VAR_INPUT
  VALUE : TIME_OF_DAY ;	//Zu prüfender Wert
  MIN : TIME_OF_DAY ;	//Zulässiger Minimalwert
  MAX : TIME_OF_DAY ;	//Zulässiger Maximalwert
END_VAR
VAR_OUTPUT
  OK : BOOL ;	//Wert im Toleranzbereich
END_VAR
BEGIN
NETWORK
TITLE =

      L     #MIN; // minmal zulässiger Wert
      L     #VALUE;
      >D    ; // falls MIN > VALUE
      SPB   NOK; // dann nicht ok
      L     #MAX;
      >D    ; // falls VALUE > MAX
      SPB   NOK; // dann nicht ok
      =     #OK; // sonst ok
      SAVE  ;
      BEA   ;
NOK:  CLR   ; // Wert nicht ok
      =     #OK;
      SAVE  ;


END_FUNCTION

FUNCTION "m7b_Scale_TOD" : TIME_OF_DAY
TITLE =Bereich Skalieren Time_Of_Day
//Skaliert eienen Wert von einem Eingagswertebereich auf einen
//Ausgangswertebereich:
//
//FC-ENO: Übersteuerungsanzeige
//
//ACHTUNG: die Eingangswerte werden nicht auf Gültigkeit geprüft
//         und der Ausgangswert wird nicht begrenzt. Bei Übersteuerung wird
//         der FC-ENO-Ausgang "1"
//
//z.B. Eingangswertebereich 100 -  300
//     Ausgangswertebereich   0 - 1000
//
//                           (MaxOutput - MinOutput)
//Xout = (Value - MinInput) --------------------------  + MinOutput
//                            (MaxInput - MinInput)
//
//
//AUTOR: Stefan Maag, Dipl.-Ing. (FH) Elektrotechnik
//DATUM: 3/2003
//INTERNET: www.maagic7.de
//
//AENDERUNGSVERMERKE:
//--------------------------------------------------------------------------------
//DATUM        NAME            AENDERUNG
//--------------------------------------------------------------------------------
//
//--------------------------------------------------------------------------------
//
//HINWEISE:
AUTHOR : 'S.Maag'
FAMILY : Maagic7
VERSION : 0.1


VAR_INPUT
  tMinInput : TIME_OF_DAY ;
  tMaxInput : TIME_OF_DAY ;
  tValue : TIME_OF_DAY ;
  tMinOutput : TIME_OF_DAY ;
  tMaxOutput : TIME_OF_DAY ;
END_VAR
VAR_TEMP
  rTemp : REAL ;
END_VAR
BEGIN
NETWORK
TITLE =Eingagswertebereich berechnen
//(MaxInput - MinInput)
      L     #tMaxInput;
      L     #tMinInput;
      -D    ; // Differenz
      DTR   ; // zu        REAL
      T     #rTemp;

NETWORK
TITLE =Faktor aus Ausgangs- und Eingangs-Wertebereich
// (MaxOutput - MinOutput)
//-------------------------
//  (MaxInput - MinInput)
      L     #tMaxOutput;
      L     #tMinOutput;
      -D    ; // Differenz
      DTR   ; // zu        REAL
      L     #rTemp;
      /R    ; // Gleitpunktdivision
      T     #rTemp;

NETWORK
TITLE =skalierter Ausgangswert
//                     (MaxOutput - MinOutput)
// (Value - MinInput) -------------------------- + MinOutput
//                      (MaxInput - MinInput)
      L     #tValue; // Eingangswert
      L     #tMinInput; // UnterGrenze Eingangswert
      -D    ; // Differenz
      DTR   ; // zu        REAL
      L     #rTemp;
      *R    ; // Gleitpunktmultiplikation
      RND   ; // zu Festpunkt 32Bit
      L     #tMinOutput;
      +D    ;
      T     #RET_VAL; // Rückgabewert
NETWORK
TITLE =FC-ENO-Ausgangs als Übersteuerungsanzeige

      L     #tMaxOutput; // MaxOutput
      >D    ; // Wert > MaxOutput
      SPB   SAVE; // Max-Wert überschritten
      TAK   ; // Ausgangswert in Akku 1 zurueck
      L     #tMinOutput;
      <D    ;
      SPB   SAVE; // MinWert unterschritten
      CLR   ;
SAVE: SAVE  ;
      CLR   ;
END_FUNCTION

FUNCTION "m7b_MinDiffABS_TOD" : VOID
TITLE =MinDiffABS_TOD: Minimale Absolutdifferenz 2er TOD-Zeiten ok!
//Überprüft, ob die absolute Differenz (absolut) zweier Time_Of_Day-Zeiten dem
//angebegenen Mindestwert entspricht. Wenn ja, dann wird ENO=True
//
//ACHTUNG: Die Differenz kann nicht im TimeOfDay-Format angeben werden, diese
//         muss TIME sein
//
//BENÖTIGTE SFCs: keine
//
//AUTOR: Stefan Maag, Dipl.-Ing. (FH) Elektrotechnik
//DATUM: 8/2008
//INTERNET: www.maagic7.de
//
//AENDERUNGSVERMERKE:
//--------------------------------------------------------------------------------
//DATUM        NAME        AENDERUNG
//--------------------------------------------------------------------------------
//
//--------------------------------------------------------------------------------
//
//HINWEISE:
AUTHOR : 'S.Maag'
FAMILY : Maagic7
VERSION : 0.1


VAR_INPUT
  TOD1 : TIME_OF_DAY ;
  TOD2 : TIME_OF_DAY ;
  MinTimeDiff : TIME ;
END_VAR
VAR_TEMP
  aktSysTime : TIME ;	//aktuelle Systemzeit
END_VAR
BEGIN
NETWORK
TITLE =prüfen ob Zeit abgelaufen ist

      L     #TOD1;
      L     #TOD2;
      -D    ;
      SPP   pos;
      NEGD  ;
pos:  L     #MinTimeDiff;
      >=D   ;
      SAVE  ;

END_FUNCTION

FUNCTION "m7b_ChangeEvent_DATE" : VOID
TITLE =Ereignis Date Wert hat sich geändert
//Der FC-ENO-Ausgang wird für einen Zyklus "1", wenn der sich der Eingangswert
//geändert hat, ansonsten ist der FC-ENO-Ausgang "0"
//
//AUTOR: Stefan Maag, Dipl.-Ing. (FH) Elektrotechnik
//DATUM: 5/2010
//INTERNET: www.maagic7.de
//
//AENDERUNGSVERMERKE:
//--------------------------------------------------------------------------------
//DATUM        NAME            AENDERUNG
//--------------------------------------------------------------------------------
//05.2010      S.Maag          Entstand aus FC150 ChangeEventTOD
//--------------------------------------------------------------------------------
//
//HINWEISE:
AUTHOR : 'S.Maag'
FAMILY : Maagic7
VERSION : 0.1


VAR_INPUT
  inDate : DATE ;
END_VAR
VAR_IN_OUT
  memDate : DATE ;
END_VAR
BEGIN
NETWORK
TITLE =

      L     #inDate; // Eingangwert
      L     #memDate; // letzter Wert
      <>D   ; // ungleich!
      SAVE  ; // als ENO ausgeben
      SPB   do; // und neuen
      BEA   ;
do:   L     #inDate; // Wert speichern
      T     #memDate;

END_FUNCTION

FUNCTION "m7b_ChangeEvent_BYTE" : VOID
TITLE =Ereignis Byte Wert hat sich geändert
//Der FC-ENO-Ausgang wird für einen Zyklus "1", wenn der sich der Eingangswert
//geändert hat, ansonsten ist der FC-ENO-Ausgang "0"
//
//AUTOR: Stefan Maag, Dipl.-Ing. (FH) Elektrotechnik
//DATUM: 8/2008
//INTERNET: www.maagic7.de
//
//AENDERUNGSVERMERKE:
//--------------------------------------------------------------------------------
//DATUM        NAME            AENDERUNG
//--------------------------------------------------------------------------------
//
//--------------------------------------------------------------------------------
//
//HINWEISE:
AUTHOR : 'S.Maag'
FAMILY : Maagic7
VERSION : 0.1


VAR_INPUT
  inBYTE : BYTE ;
END_VAR
VAR_IN_OUT
  memBYTE : BYTE ;
END_VAR
BEGIN
NETWORK
TITLE =

      L     #inBYTE; // Eingangwert
      L     #memBYTE; // letzter Wert
      <>I   ; // ungleich!
      SAVE  ; // als ENO ausgeben
      SPB   do; // und neuen
      BEA   ;
do:   L     #inBYTE; // Wert speichern
      T     #memBYTE;

END_FUNCTION

FUNCTION "m7b_ByteCompare" : VOID
TITLE =BYTE Compare : 2 Bytes vergleichen
//Der FC-ENO-Ausgang wird True, wenn Byte1=Byte2
//
//AUTOR: Stefan Maag, Dipl.-Ing. (FH) Elektrotechnik
//DATUM: 4/2009
//INTERNET: www.maagic7.de
//
//AENDERUNGSVERMERKE:
//--------------------------------------------------------------------------------
//DATUM        NAME            AENDERUNG
//--------------------------------------------------------------------------------
//
//--------------------------------------------------------------------------------
//
//HINWEISE:
AUTHOR : 'S.Maag'
FAMILY : Maagic7
VERSION : 0.1


VAR_INPUT
  Byte1 : BYTE ;
  Byte2 : BYTE ;
END_VAR
BEGIN
NETWORK
TITLE =

      L     #Byte1;
      L     #Byte2;
      ==I   ;
      SAVE  ;
      CLR   ;
END_FUNCTION

FUNCTION "m7b_SPLIT_BYTE_TO_8xINT" : VOID
TITLE =Splits 1 Byte (8xFLAGs) into 8xINT
//AUTOR: Stefan Maag, Dipl.-Ing. (FH) Elektrotechnik
//DATUM: 11/2012
//INTERNET: www.maagic7.de
//
//AENDERUNGSVERMERKE:
//--------------------------------------------------------------------------------
//DATUM        NAME        AENDERUNG
//--------------------------------------------------------------------------------
//
//--------------------------------------------------------------------------------
//
//HINWEISE:
AUTHOR : 'S.Maag'
FAMILY : Maagic7
VERSION : 0.1


VAR_INPUT
  FLAGs : BYTE ;	//Byte: FLAGs
END_VAR
VAR_OUTPUT
  INT_BIT_0 : INT ;
  INT_BIT_1 : INT ;
  INT_BIT_2 : INT ;
  INT_BIT_4 : INT ;
  INT_BIT_3 : INT ;
  INT_BIT_5 : INT ;
  INT_BIT_6 : INT ;
  INT_BIT_7 : INT ;
END_VAR
VAR_TEMP
  wADR : WORD ;
  LOOPS : INT ;
END_VAR
BEGIN
NETWORK
TITLE =

      L     P##INT_BIT_0; // load AR1 with Pointer
      LAR1  ; // of first INT output

NETWORK
TITLE =

      L     #FLAGs;
      L     8; // Schleifenzähler
LOOP: T     #LOOPS;
      TAK   ; // FLAGs back to AKKU 1
      SRW   1;
      SPP   Hi;
      L     0;
      SPA   save;
Hi:   L     1;
save: T     W [AR1,P#0.0];
      +AR1  P#2.0;
      TAK   ; // FLAGs back to AKKU 1
      L     #LOOPS; // Schleifenzähler laden
      LOOP  LOOP; // Schleife bearbeiten
END_FUNCTION

FUNCTION_BLOCK "cPUMP"
TITLE =Pumpensteuerung mit Min- Laufzeit und Impulsbetrieb
//Pumpensteuerung mit Minimallaufzeit sowie Impulsbetrieb (Sommerbetrieb)
//AUTOR: Stefan Maag, Dipl.-Ing. (FH) Elektrotechnik
//DATUM: 7/2012
//
//AENDERUNGSVERMERKE:
//--------------------------------------------------------------------------------
//DATUM        NAME        AENDERUNG
//--------------------------------------------------------------------------------
//
//--------------------------------------------------------------------------------
//
//HINWEISE:
AUTHOR : 'S.Maag'
FAMILY : Maagic7
VERSION : 0.1


VAR_INPUT
  FRG : BOOL ;	//Freigabe
  START : BOOL ;	//Pumpe Start
  cfg_PulsBetrieb : BOOL ;	//Pulsbetrieb: nach Max. Ausschaltzeit timPulsOn einschalten
  timMinOn : TIME ;	//Mindestlaufzeit
  timMinOFF : TIME ;	//Min Ausschaltzeit
  timMaxOFF : TIME ;	//Max Ausschaltzeit
  timPulsON : TIME ;	//Einschaltpuls nach max. Ausschaltzeit
END_VAR
VAR_OUTPUT
  PUMP : BOOL ;
END_VAR
VAR
  Q_TON_Min : BOOL ;
  Q_PUMP : BOOL ;
  Q_TON_MaxOff : BOOL ;
  Q_PULS_ON : BOOL ;
  Q_TOF_MinAus : BOOL ;
  TON_MinON : "TON";
  ton_maxOff : "TON";
END_VAR
VAR_TEMP
  fktMinON : BOOL ;
  MinAusSperre : BOOL ;
  dummy : BOOL ;
  tMinOn : TIME ;
  tOFF : TIME ;
  DSP_tOFF : TIME ;
END_VAR
BEGIN
NETWORK
TITLE =



NETWORK
TITLE =Funktion Mindeslaufzeit aktiv

      L     #timMinOn;
      L     0;
      <>D   ;
      =     #fktMinON;
NETWORK
TITLE =(tMaxOff > tMinOff)? sonst tMinOff verwenden

      L     #timMaxOFF;
      L     #timMinOFF;
      >=D   ;
      =     L     14.0;
      U     L     14.0;
      SPBNB _001;
      L     #timMaxOFF;
      T     #tOFF;
_001: NOP   0;
      U     L     14.0;
      NOT   ;
      SPBNB _002;
      L     #timMinOFF;
      T     #tOFF;
_002: NOP   0;
NETWORK
TITLE =Maximale Ausschaltzeit

      U(    ;
      UN    #Q_PUMP;
      =     L     14.0;
      BLD   103;
      CALL #ton_maxOff (
           IN                       := L     14.0,
           PT                       := #tOFF,
           Q                        := #Q_TON_MaxOff,
           ET                       := #DSP_tOFF);
      U     BIE;
      )     ;
      U     #Q_TON_MaxOff;
      U     #cfg_PulsBetrieb;
      S     #Q_PULS_ON;
      U(    ;
      ON    #Q_TON_Min;
      ON    #FRG;
      )     ;
      R     #Q_PULS_ON;
      NOP   0;
NETWORK
TITLE =Mindestauschaltzeit Sperre
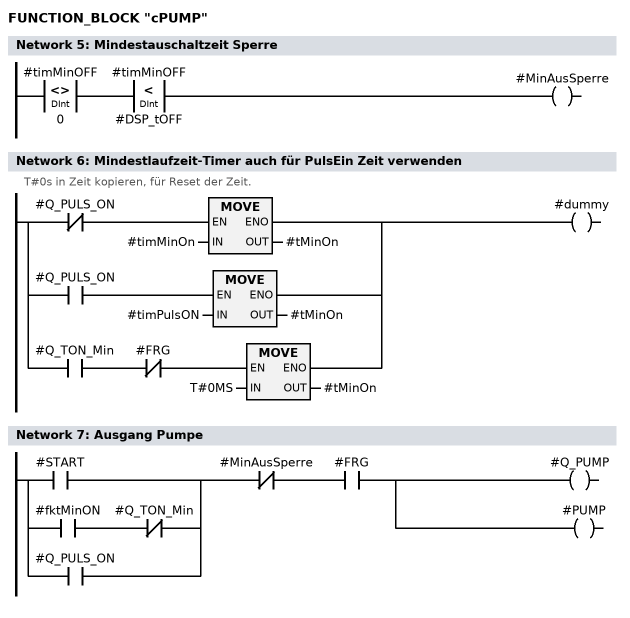

      U(    ;
      L     #timMinOFF;
      L     0;
      <>D   ;
      )     ;
      U(    ;
      L     #timMinOFF;
      L     #DSP_tOFF;
      <D    ;
      )     ;
      =     #MinAusSperre;
NETWORK
TITLE =Mindestlaufzeit-Timer auch für PulsEin Zeit verwenden
//T#0s in Zeit kopieren, für Reset der Zeit.
//
      O(    ;
      UN    #Q_PULS_ON;
      SPBNB _003;
      L     #timMinOn;
      T     #tMinOn;
      SET   ;
      SAVE  ;
      CLR   ;
_003: U     BIE;
      )     ;
      O(    ;
      U     #Q_PULS_ON;
      SPBNB _004;
      L     #timPulsON;
      T     #tMinOn;
      SET   ;
      SAVE  ;
      CLR   ;
_004: U     BIE;
      )     ;
      O(    ;
      U     #Q_TON_Min;
      UN    #FRG;
      SPBNB _005;
      L     T#0MS;
      T     #tMinOn;
      SET   ;
      SAVE  ;
      CLR   ;
_005: U     BIE;
      )     ;
      =     #dummy;
NETWORK
TITLE =Ausgang Pumpe

      U(    ;
      O     #START;
      O     ;
      U     #fktMinON;
      UN    #Q_TON_Min;
      O     #Q_PULS_ON;
      )     ;
      UN    #MinAusSperre;
      U     #FRG;
      =     #Q_PUMP;
      =     #PUMP;
NETWORK
TITLE =Pumpensignal auch auf ENO-Ausgang

      U     #Q_PUMP;
      SAVE  ;

END_FUNCTION_BLOCK

FUNCTION "m7b_RP_BIT_WRITE" : VOID
TITLE =Ringpuffer schreiben BIT (0..255) (32 Bytes)
//AUTOR: Stefan Maag, Dipl.-Ing. (FH) Elektrotechnik
//DATUM: 05/2003
//INTERNET: www.maagic7.de
//
//AENDERUNGSVERMERKE:
//--------------------------------------------------------------------------------
//DATUM        NAME            AENDERUNG
//--------------------------------------------------------------------------------
//09.10.2010   S.Maag          Aufnahme des Bausteins in Maagic7
//                             von DBNr auf BlockDB umgestellt
//--------------------------------------------------------------------------------
//
//HINWEISE:
AUTHOR : 'S.Maag'
FAMILY : Maagic7
VERSION : 0.1


VAR_INPUT
  DB_RP : BLOCK_DB ;	//Datenbaustein Ringpuffer
  StartAdrByte : INT ;	//Startadresse Byte des Ringpuffers im DB
  SIGNAL : BOOL ;	//Eingang des zu speichernden Signals
  FLKp : BOOL ;	//positive Flanke Schreibtakt
  FLKn : BOOL ;	//negative Flanke Schreibtakt
END_VAR
VAR_IN_OUT
  RP_POINTER : INT ;
END_VAR
VAR_TEMP
  tmpDB : INT ;
END_VAR
BEGIN
NETWORK
TITLE =

      U     #FLKp; // positive Flanke Schreibsignal
      SPB   P;

      U     #FLKn; // negative Flanke Schreibsignal
      SPB   N;

      CLR   ; // ENO = FALSE, => keine Verarbeitung
      SAVE  ;
      BEA   ;

P:    L     #RP_POINTER; // Pointer vorwärts zählen
      INC   1; // INC: Bytebefehl 0..255
      SPA   save;

N:    L     #RP_POINTER; // Pointer rückwärts zählen
      DEC   1; // DEC: Bytebefehl 0..255

save: T     #RP_POINTER; // neuen Pointer speichern
      SET   ;
      SAVE  ; // ENO = TRUE, => Verarbeitung
      CLR   ;


NETWORK
TITLE =DB öffnen und Pointer auf aktuelles Bit in AR1
//Adressregister 1 retten ist nöchtig, da dies automatisch bei Bausteinaufrufen
//mit CALL geschieht (UC Aufrufe sichern nicht!)
      AUF   #DB_RP;

      L     #StartAdrByte; // StartAdr. ins BitPointerFormat
      SLD   3;
      L     #RP_POINTER; // Nr des akt. Bits
      +D    ; // Pointer auf aktuelles Bit
      L     P#0.0; // Nullpointer addieren für Pointerkennung
      +D    ;
      LAR1  ;
NETWORK
TITLE =Signalzustand in Ringpuffer schreiben

      U     #SIGNAL;
      =     DBX [AR1,P#0.0]; // Pointer auf aktuelles Bit

END_FUNCTION

FUNCTION "m7b_RB_BIT_READ" : VOID
TITLE =Ringpuffer lesen BIT (0..255) (32 Bytes)
//AUTOR: Stefan Maag, Dipl.-Ing. (FH) Elektrotechnik
//DATUM: 05/2003
//INTERNET: www.maagic7.de
//
//AENDERUNGSVERMERKE:
//--------------------------------------------------------------------------------
//DATUM        NAME            AENDERUNG
//--------------------------------------------------------------------------------
//09.10.2010   S.Maag          Aufnahme des Bausteins in Maagic7
//                             von DBNr auf BlockDB umgestellt
//--------------------------------------------------------------------------------
//
//HINWEISE:
AUTHOR : 'S.Maag'
FAMILY : Maagic7
VERSION : 0.1


VAR_INPUT
  DB_RP : BLOCK_DB ;	//Datenbaustein Ringpuffer
  StartAdrByte : INT ;	//StartAdresseByte des RingPuffers (Länge = 32 Byte)
  RP_POINTER : INT ;	//aktueller RingpufferPointer
  DISTANZ : INT ;	//Distanz des auszulesenden Wertes
END_VAR
VAR_OUTPUT
  BIT : BOOL ;
END_VAR
VAR_TEMP
  AR1 : DWORD ;
END_VAR
BEGIN
NETWORK
TITLE =DB öffnen und Pointer auf aktuelles Bit in AR1

      TAR1  #AR1; // Adressregister 1 sichern

      AUF   #DB_RP;

      L     #RP_POINTER; // Nr des akt. Bits
      L     #DISTANZ; // Auslesedistanz
      -I    ; // Auslesepositon berechnen
      L     255; // Berechnung auf ByteFormat
      UW    ; // begrenzen (geht leider nicht mit DEC)
      L     #StartAdrByte; // StartAdr. ins Pointerformat
      SLD   3;
      +D    ; // Pointer auf aktuelles Bit
      L     P#0.0; // Nullpointer addieren für Pointerkennung
      +D    ;
      LAR1  ;
NETWORK
TITLE =Signalzustand aus Ringpuffer lesen

      U     DBX [AR1,P#0.0]; // Pointer auf aktuelles Bit
      =     #BIT;

      TAR1  #AR1; // Adressregister 1 sichern
END_FUNCTION

FUNCTION "m7b_RingBuffer_ptr_INC" : INT
TITLE =Ringpuffer Pointer addieren (Pointeroffset und Auslesepos.)
//AUTOR: Stefan Maag, Dipl.-Ing. (FH) Elektrotechnik
//DATUM: 07/2010
//INTERNET: www.maagic7.de
//
//AENDERUNGSVERMERKE:
//--------------------------------------------------------------------------------
//DATUM        NAME            AENDERUNG
//--------------------------------------------------------------------------------
//
//--------------------------------------------------------------------------------
//
//HINWEISE:
AUTHOR : 'S.Maag'
FAMILY : Maagic7
VERSION : 0.1


VAR_INPUT
  RP_POINTER : INT ;	//Pointer Ringpuffer 0..255
  RP_OFFSET : INT ;	//Pointer Rinpuffer Offset (0.255)
END_VAR
BEGIN
NETWORK
TITLE =

      SET   ;
      SAVE  ;
      CLR   ;

NETWORK
TITLE =

      L     #RP_POINTER; // Pointer 1 Ringpuffer
      L     #RP_OFFSET; // Pointer Offset bzw. Pointer 2
      +I    ; // Pointer addieren
      L     255; // auf Byte begrenzen
      UW    ;
      T     #RET_VAL; // Summe Pointer 0..255


END_FUNCTION

FUNCTION "m7b_RingBuffer_ptr_DEC" : INT
TITLE =Ringpuffer Pointer subtrahieren (Pointeroffset und Auslesepos.)
//AUTOR: Stefan Maag, Dipl.-Ing. (FH) Elektrotechnik
//DATUM: 07/2010
//INTERNET: www.maagic7.de
//
//AENDERUNGSVERMERKE:
//--------------------------------------------------------------------------------
//DATUM        NAME            AENDERUNG
//--------------------------------------------------------------------------------
//
//--------------------------------------------------------------------------------
//
//HINWEISE:
AUTHOR : 'S.Maag'
FAMILY : Maagic7
VERSION : 0.1


VAR_INPUT
  RP_POINTER : INT ;	//Pointer Ringpuffer 0..255
  RP_OFFSET : INT ;	//Pointer Rinpuffer Offset (0.255)
END_VAR
BEGIN
NETWORK
TITLE =

      SET   ;
      SAVE  ;
      CLR   ;

NETWORK
TITLE =

      L     #RP_POINTER; // Pointer 1 Ringpuffer
      L     #RP_OFFSET; // Pointer Offset bzw. Pointer 2
      -I    ; // Pointer subtrahieren
      L     255; // auf Byte begrenzen
      UW    ;
      T     #RET_VAL; // Summe Pointer 0..255


END_FUNCTION

FUNCTION "m7b_X_SWITCH_BIT" : VOID
TITLE =Cross Swtich for Bit's
//Cross Switch for BIT's
//
//[IN]
//X     : Switch command: LO: 1:1 D1_1=DO1; HI: 1X1 DI_1=DO_2
//DI_1  : Digitial IN 1
//DI_2  : Digitial IN 2
//
//[OUT]
//DO_1  : Digital Out 1
//DO_2  : Digital Out 2
//
//[FC-ENO]  :
//
//
//AUTOR: Stefan Maag, Dipl.-Ing. (FH) Elektrotechnik
//DATUM: 6/2012
//INTERNET: www.maagic7.de
//
//AENDERUNGSVERMERKE:
//--------------------------------------------------------------------------------
//DATUM        NAME            AENDERUNG
//--------------------------------------------------------------------------------
//
//--------------------------------------------------------------------------------
//
//HINWEISE:
AUTHOR : 'S.Maag'
FAMILY : Maagic7
VERSION : 0.1


VAR_INPUT
  X : BOOL ;	//Switch command: LO: 1:1 D1_1=DO1; HI: DI_1=DO_2
  DI_1 : BOOL ;	//Digitial IN 1
  DI_2 : BOOL ;	//Digitial IN 2
END_VAR
VAR_OUTPUT
  DO_1 : BOOL ;	//Digital Out 1
  DO_2 : BOOL ;	//Digital Out 2
END_VAR
BEGIN
NETWORK
TITLE =

      SET   ;
      SAVE  ;
      CLR   ;

NETWORK
TITLE =

      U     #X;
      SPB   xed;

      U     #DI_1;
      =     #DO_1;

      U     #DI_2;
      =     #DO_2;
      BEA   ;

xed:  U     #DI_1;
      =     #DO_2;

      U     #DI_2;
      =     #DO_1;


END_FUNCTION

FUNCTION "m7d_TimeEventDay_DEZ" : VOID
TITLE =TimeEventDay
//Funktion zum Erzeugen eines Ereignisses zu einer bestimmten Zeit. Der
//Ereignismerker muß nach der Verarbeitung extern zurückgesetzt werden.
//Durch die Verwendung eines Hilfsmerkers wird garantiert, daß das Ereignis
//bei sofortiger Verarbeitung und rücksetzen des Ereignismerkers, nicht direkt
//wieder ausgelöst wird.
//
//[IN]
//HOUR : Stunde
//MIN  : Minute
//SEC  : Sekunde
//
//[INOUT]
//EVENT    : Ereignismerker (muß nach Verarbeitung extern gelöscht werden)
//HM_EVENT : benötigter Hilfsmerker
//BENÖTIGTE SFCs: SFC1 - READ_CLK
//
//AUTOR: Stefan Maag, Dipl.-Ing. (FH) Elektrotechnik
//DATUM: 9/2004
//INTERNET: www.maagic7.de
//
//AENDERUNGSVERMERKE:
//--------------------------------------------------------------------------------
//DATUM        NAME        AENDERUNG
//--------------------------------------------------------------------------------
//
//--------------------------------------------------------------------------------
//
//HINWEISE:
AUTHOR : 'S.Maag'
FAMILY : Maagic7
VERSION : 0.1


VAR_INPUT
  HOUR : INT ;
  MIN : INT ;
  SEC : INT ;
END_VAR
VAR_IN_OUT
  EVENT : BOOL ;	//Ereignis-Merker (wird gesetzt)
  HM : BOOL ;	//Hilfsmerker
END_VAR
VAR_TEMP
  DATE_TIME : DATE_AND_TIME ;
  ERR_CODE : INT ;
  m_STD : INT ;
  m_MIN : INT ;
  m_SEC : INT ;
END_VAR
BEGIN
NETWORK
TITLE =Zeit in temporäreren Variablenbereich einlesen

      CALL "READ_CLK" (
           RET_VAL                  := #ERR_CODE,
           CDT                      := #DATE_TIME);
      NOP   0;
NETWORK
TITLE =Stunden, Minuten und Sekunden aus DATE_AND_TIME extrahieren
//Das DATE_AND_TIME Format benötigt 8 Byte im BCD-Format
//Der Wertebereich geht von DT#1990-1-1-0:0:0.0 bis DT#2089-12-31-23:59:59.999
//
//BYTE 0:  Jahr
//BYTE 1:  Monat
//BYTE 2:  Tag
//BYTE 3:  Stunde
//BYTE 4:  Minute
//BYTE 5:  Sekunde
//BYTE 6:  100er und 10er Stelle von Millisekunden
//BYTE 7:  Bit 4..7: 1er  Stelle von Millisekunden
//BYTE 7:  Bit 0..3: Wochentag (1=Sonntag, 2=Montag, ..., 7=Samstag)
      L     LB     3; // Stunde
      BTI   ;
      T     #m_STD;

      L     LB     4; // Minute
      BTI   ;
      T     #m_MIN;

      L     LB     5; // Sekunde
      BTI   ;
      T     #m_SEC;


NETWORK
TITLE =Zeit prüfen und Event erzeugen


      L     #HOUR;
      L     #m_STD;
      <>I   ; // Stunde stimmt nicht, dann Ende
      SPB   END;

      L     #MIN;
      L     #m_MIN;
      <>I   ; // Minute stimmt nicht
      R     #HM; // HM wieder löschen
      SPB   END;

      L     #SEC; // Wenn die Sekunden erreicht bzw. überschritten sind,
      L     #m_SEC; // dann Ereignis auslösen
      >=I   ;
      UN    #HM;
      S     #HM;
      S     #EVENT;
      SPA   END;

END:  U     #EVENT; // Ereignis als FC_ENO ausgeben, für direkte Weiterverschaltung und Status
      SAVE  ;
      CLR   ;
END_FUNCTION

FUNCTION_BLOCK "m7b_SRK_AUSRICHTEN"
TITLE =Standardablauf für Ausrichtfunktion mit Zylinder
//- Ausfahren bis Endstellung
//- Zeit warte
//- Einfahren bis Grundstellung
//- READY
AUTHOR : 'S.Maag'
FAMILY : Maagic7
VERSION : 0.1


VAR_INPUT
  START : BOOL ;
  RESET : BOOL ;
  POS_AST : BOOL ;
  POS_GST : BOOL ;
  timDelayAST : TIME ;
END_VAR
VAR_OUTPUT
  CMD_AST : BOOL ;
  CMD_GST : BOOL ;
  MSG_RUN : BOOL ;
  MSG_READY : BOOL ;
  DSP_SNR : INT ;
END_VAR
VAR
  SNR : INT ;
  timTimer : TIME ;
  TON_TIMER : "TON";
  Q_TIMER : BOOL ;
  START_TIMER : BOOL ;
  HM_FP_START : BOOL ;
END_VAR
VAR_TEMP
  tmpDSP_TIMER : TIME ;
END_VAR
BEGIN
NETWORK
TITLE =



NETWORK
TITLE =Timer auf mindestens 1ms begrenzen, sonst startet Zeit nicht!

      L     #timTimer;
      L     T#1MS;
      >=D   ;
      SPB   ne2;
      T     #timTimer;
ne2:  NOP   0;
NETWORK
TITLE =Timer für Verzögerungen

      CALL #TON_TIMER (
           IN                       := #START_TIMER,
           PT                       := #timTimer,
           Q                        := #Q_TIMER,
           ET                       := #tmpDSP_TIMER);

NETWORK
TITLE =Schrittablauf clr

      U     #RESET; // Schrittabläufe clr
      SPBNB _001;
      L     0;
      T     #SNR;
_001: NOP   0;
NETWORK
TITLE =Standard Ablaufsteuerung mit INIT und CLR-Zweig


      L     #SNR; // Schrittnummer
      SPL   CLR; // Sprungziel bei SNR>max
      SPA   INIT; // 0-Schritt, Initialisierung
      SPA   S1; // Startschritt
      SPA   S2;
      SPA   S3;
      SPA   S4;
//      SPA   S5
//      SPA   S6

CLR:  SET   ; // CLR Aktionsmerker die über das Ende der Schrittkette nicht mehr benötigt werden
      R     #START_TIMER;
      R     #MSG_RUN;

      L     1; // Schrittnummer
      T     #SNR; // auf Startschritt stellen
      T     #DSP_SNR; // Schrittnummer Anzeige
      SPA   END;

INIT: SET   ; // Initalisierung
      R     #MSG_READY;

// hier die bei INIT zu löschenden Merker eintragen
// z.B. Aktionsmerker die über das Ende der Schrittkette weiterhin benötigt werden
// wird bei verketteten oder mehrstufigen Schrittabläufen benötigt
      CLR   ;
      SPA   CLR;
      SPA   SET; // wird nur benötigt, damit die Entwicklungsumgebung die Sprungmarke nicht löscht


NETWORK
TITLE =Schrittweiterschaltung, bzw. Bausteinende

NEXT: L     #SNR; // NEXT : Schrittnummer auf nächsten
      +     1; // Schritt
SET:  T     #SNR; // Ablauf auf Schritt mit Nr. in Akku 1 setzen

END:  L     #SNR; // Sprungmarke für Baustein ENDE
      T     #DSP_SNR; // Schrittnummer Anzeige
      L     1; // Wenn Ablauf läuft, dann ENO-Ausgang = 1
      >I    ;
      SAVE  ;
      CLR   ;
      BEA   ;

NETWORK
TITLE =Startschritt

S1:   U     #START; // Start ausrichten
      FP    #HM_FP_START;
      S     #MSG_RUN;
      R     #MSG_READY;
      S     #CMD_AST;
      R     #CMD_GST;
      SPB   NEXT;
      SPA   END;
NETWORK
TITLE =Schritt 2: Enstellung erreicht? Timer starten!

S2:   U     #POS_AST;
      SPBN  END;

      S     #START_TIMER; // Timer starten
      L     #timDelayAST; // Zeit für Timer
      T     #timTimer;

      SPA   NEXT;

NETWORK
TITLE =Schritt 3: Timer abgelaufen? zu Grundstellung!

S3:   U     #Q_TIMER; // Timer abgelaufen
      R     #START_TIMER;
      R     #CMD_AST;
      S     #CMD_GST;
      SPB   NEXT;
      SPA   END;

NETWORK
TITLE =Schritt 4: Grundstellung erreicht? READY!

S4:   U     #POS_GST;
      S     #MSG_READY;
      SPB   NEXT;
      SPA   END;

END_FUNCTION_BLOCK

FUNCTION "m7b_TOL_HYS_INT" : VOID
TITLE =Position mit Toleranzen und Hysteres prüfen [INT]
//Anwendung:
//Toleranzprüfungen bei welchen das ok-Signal erst bei überschreiten
//einer größeren Toleranz wieder gelöscht werden soll
//
//z.B. Positionieranwendungen: nachpositionieren erst wenn Hysterseschwelle
//der Toleranz überschritten ist
//
//AUTOR: Stefan Maag, Dipl.-Ing. (FH) Elektrotechnik
//DATUM: 01/2015
//INTERNET: www.maagic7.de
//
//AENDERUNGSVERMERKE:
//--------------------------------------------------------------------------------
//DATUM        NAME        AENDERUNG
//--------------------------------------------------------------------------------
//
//--------------------------------------------------------------------------------
//
//HINWEISE:
AUTHOR : 'S.Maag'
FAMILY : Maagic7
VERSION : 0.1


VAR_INPUT
  IST : INT ;	//Istwert Achse
  SOLL : INT ;	//Sollwert
  TOL : INT ;	//Toleranz Posiitionierung Achse Stop
  HYS : INT ;	//Hysterese, Position nicht mehr o.k.
END_VAR
VAR_IN_OUT
  io_OK : BOOL ;
END_VAR
VAR_TEMP
  TOL_HYS : INT ;
  TOL_1_OK : BOOL ;
  TOL_2_OK : BOOL ;
END_VAR
BEGIN
NETWORK
TITLE =Position mit Toleranzen und Hysterese prüfen

      L     #TOL; // Toleranz
      L     #HYS; // Hysteres
      +I    ;
      T     #TOL_HYS; // Toleranz, Hystereseschwelle

      L     #SOLL; // aktuelle Sollposition
      L     #IST; // aktuelle Istposition
      -I    ; // Positionierdifferenz
      SPP   PLUS;
      NEGI  ; // nach positiv

PLUS: L     #TOL; // Toleranz für Position ok
      <=I   ;
      S     #io_OK; // Ausgang Position ok
      TAK   ; // Positionsdifferenz in AKKU1
      L     #TOL_HYS; // Toleranz für Positionierung
      >I    ;
      R     #io_OK; // Ausgang Position ok

      U     #io_OK;
      SAVE  ;
      CLR   ;


END_FUNCTION

FUNCTION "m7b_AVG_MIN_MAX_4xINT" : VOID
TITLE =MIN, MAX, AVERAGE from activated channels (CH1,CH2,CH3,CH4)
//Give back the minimum, maximum and average value of 4 values (channels)
//
//INPUT:
//iCH1      : value channel 1
//iCH2      : value channel 2
//iCH3      : value channel 3
//iCH4      : value channel 4
//iCH_OFF   : value is all channels are deactivated (OFF)
//
//CH1_active: FLASE: channel is deactivated (not included in calcuation)
//.           TRUE : channel is activated (included in calculation)
//.
//CH4_active:
//
//---------------------------------------------------------
//OUTPUT:
//AVG       : AVERAGE(CH1,CH2,CH3,CH4) or CH_off if all channels deactivated
//MIN       : MINIMUM(CH1,CH2,CH3,CH4) or CH_off if all channels deactivated
//MAX       : MAXIMUM(CH1,CH2,CH3,CH4) or CH_off if all channels deactivated
//NoCH_min  : Channel No. of minimum value; 0 if all channels deactivated
//NoCH_max  : Channel No. of maximum value; 0 if all channels deactivated
//NoOfActCH : Number of activated channels [0..4]
//FC-ENO    : FALSE: alle channels are disactivated; CH_OFF is selected
//            TRUE : at least 1 channel is activated; Min/Max is selected
//
//
//AUTOR: Stefan Maag, Dipl.-Ing. (FH) Elektrotechnik
//DATUM: 8/2018
//
//AENDERUNGSVERMERKE:
//--------------------------------------------------------------------------------
//DATUM        NAME      AENDERUNG
//--------------------------------------------------------------------------------
//06.08.2018   S.Maag    created by editing FC233 m7b_AVG_MIN_MAX_4xREAL
//24.09.2015   S.Maag    Function tested i.o.
//--------------------------------------------------------------------------------
//
//HINWEISE:
AUTHOR : 'S.Maag'
FAMILY : Maagic7
VERSION : 0.1


VAR_INPUT
  iCH1 : INT ;	//Value channel 1
  iCH2 : INT ;	//Value channel 2
  iCH3 : INT ;	//Value channel 3
  iCH4 : INT ;	//Value channel 4
  iCH_OFF : INT ;	//Value if all channels are deactivated
  CH1_active : BOOL ;	//TRUE activates channel l
  CH2_active : BOOL ;	//TRUE activates channel 2
  CH3_active : BOOL ;	//TRUE activates channel 3
  CH4_active : BOOL ;	//TRUE activates channel 4
END_VAR
VAR_OUTPUT
  iAVG : INT ;	//Average value
  iMIN : INT ;	//Minimum value
  iMAX : INT ;	//Maximum value
  iNoCH_min : INT ;	//Channel No of Min Value (1..3) or 0 if all channels are OFF
  iNoCH_max : INT ;	//Channel No of Max Value (1..3) or 0 if all channels are OFF
  iNoOfActCH : INT ;	//Number of activated channel [0..4]
END_VAR
VAR_TEMP
  off : BOOL ;
  tmpNoOfCHs : INT ;
  ARY : ARRAY  [1 .. 4 ] OF STRUCT
   iVAL : INT ;
   iCH : INT ;
   CHisActive : BOOL ;
  END_STRUCT ;
  tmpMin : STRUCT
   iVAL : INT ;
   iCH : INT ;
   IsValid : BOOL ;
  END_STRUCT ;
  tmpMax : STRUCT
   iVAL : INT ;
   iCH : INT ;
   IsValid : BOOL ;
  END_STRUCT ;
END_VAR
BEGIN
NETWORK
TITLE =



NETWORK
TITLE =move activated channels to a temp. ARRAY & count active channels
//if a channel is not activated, it's temporary variable will be 0.0
      L     0; // clear temporary channel variables
      T     #ARY[1].iVAL;
      T     #ARY[2].iVAL;
      T     #ARY[3].iVAL;
      T     #ARY[4].iVAL;

      L     0; // clear the channel no.
      T     #tmpNoOfCHs;
      T     #ARY[1].iCH;
      T     #ARY[2].iCH;
      T     #ARY[3].iCH;
      T     #ARY[4].iCH;

      CLR   ;
      =     #ARY[1].CHisActive;
      =     #ARY[2].CHisActive;
      =     #ARY[3].CHisActive;
      =     #ARY[4].CHisActive;

      UN    #CH1_active; // copy CH1 if activated
      SPB   chk2;

      S     #ARY[1].CHisActive;
      L     #iCH1;
      T     #ARY[1].iVAL;
      L     1;
      T     #ARY[1].iCH;

      L     #tmpNoOfCHs;
      INC   1;
      T     #tmpNoOfCHs;

chk2: UN    #CH2_active; // copy CH2 if activated
      SPB   chk3;

      S     #ARY[2].CHisActive;
      L     #iCH2;
      T     #ARY[2].iVAL;
      L     2;
      T     #ARY[2].iCH;

      L     #tmpNoOfCHs;
      INC   1;
      T     #tmpNoOfCHs;


chk3: UN    #CH3_active; // copy CH3 if activated
      SPB   chk4;

      S     #ARY[3].CHisActive;
      L     #iCH3;
      T     #ARY[3].iVAL;
      L     3;
      T     #ARY[3].iCH;

      L     #tmpNoOfCHs;
      INC   1;
      T     #tmpNoOfCHs;


chk4: UN    #CH4_active; // copy CH4 if activated
      SPB   ne3;

      S     #ARY[4].CHisActive;
      L     #iCH4;
      T     #ARY[4].iVAL;
      L     4;
      T     #ARY[4].iCH;

      L     #tmpNoOfCHs;
      INC   1;
      T     #tmpNoOfCHs;

ne3:  NOP   0;
NETWORK
TITLE =Check: all channels OFF

      L     #tmpNoOfCHs;
      T     #iNoOfActCH; // FC Output: Number of active channels
      L     0;
      ==I   ;
      =     #off;
      NOT   ;
      SAVE  ; // ENO=FALSE if all channels are deactivated
      CLR   ;

NETWORK
TITLE =AVAERAGE (CH1, CH2, CH3, CH4)
//calculate the average of CH1..4
      L     #iCH_OFF; // if all channels are deactivated,
      U     #off; // the average value is 0.0
      SPB   sAvg; // save the avarage value

      L     #ARY[1].iVAL; // building the sum of all channels
      L     #ARY[2].iVAL; // if channel is deactivated, tmp_CH-Value is 0.0
      +I    ;
      L     #ARY[3].iVAL;
      +I    ;
      L     #ARY[4].iVAL;
      +I    ; // = CH1+CH2+CH3+CH4
      L     #tmpNoOfCHs; // number of activated channels
      /I    ;
sAvg: T     #iAVG; // the AVERAGE value of all activated channels


NETWORK
TITLE =COPY first Element of ARY to tmpMin and tmpMax
//to start min/max check with first element of CH-Array, the first Array-Element
//is copied to to the tmpMin and tmpMax structure
      L     #ARY[1].iVAL;
      T     #tmpMin.iVAL;
      T     #tmpMax.iVAL;

      L     #ARY[1].iCH;
      T     #tmpMin.iCH;
      T     #tmpMax.iCH;

      U     #ARY[1].CHisActive;
      =     #tmpMin.IsValid;
      =     #tmpMax.IsValid;

NETWORK
TITLE =Get the MINIMUM value
//
//
      L     #tmpMin.iVAL; // tempMin.Val
      L     #ARY[2].iVAL; // CH2.Val
      >I    ; // IF CH2.Val < tmpMin
      U     #ARY[2].CHisActive; //    AND CH2.IsActivated
      ON    #tmpMin.IsValid; //    OR  NOT tmpMin.IsValid
      SPBN  mn3; // ELSE continue with CH3

      L     #ARY[2].iVAL; // THEN COPY CH2->tmpMin, because CH2 is the
      T     #tmpMin.iVAL; // act. minimum or tmpMin is not valid

      L     #ARY[2].iCH;
      T     #tmpMin.iCH;

      U     #ARY[2].CHisActive; // (if CH2 is not activated
      =     #tmpMin.IsValid; //  then tmpMin is not valid)

mn3:  L     #tmpMin.iVAL; // Channel 3 !see above documentation CH2!
      L     #ARY[3].iVAL;
      >I    ;
      U     #ARY[3].CHisActive;
      ON    #tmpMin.IsValid;
      SPBN  mn4;

      L     #ARY[3].iVAL;
      T     #tmpMin.iVAL;

      L     #ARY[3].iCH;
      T     #tmpMin.iCH;

      U     #ARY[3].CHisActive;
      =     #tmpMin.IsValid;

mn4:  L     #tmpMin.iVAL; // Channel 4
      L     #ARY[4].iVAL;
      >I    ;
      U     #ARY[4].CHisActive;
      ON    #tmpMin.IsValid;
      SPBN  mn5;

      L     #ARY[4].iVAL;
      T     #tmpMin.iVAL;

      L     #ARY[4].iCH;
      T     #tmpMin.iCH;

      U     #ARY[4].CHisActive;
      =     #tmpMin.IsValid;

mn5:  L     #tmpMin.iVAL; // If tmpMin.Val IsValid
      U     #tmpMin.IsValid;
      SPB   smin; // THEN copy the min. to FC-Out

      L     0; // ELSE copy 0 to FC-Out
      T     #tmpMin.iCH;
      L     #iCH_OFF;

smin: T     #iMIN; // copy the min. to FC-Out
      L     #tmpMin.iCH; // channel no. with minimum
      T     #iNoCH_min;


NETWORK
TITLE =Get the MAXIUM value

      L     #tmpMax.iVAL; // tempMax.Val
      L     #ARY[2].iVAL; // CH2.Val
      <I    ; // IF CH2.Val > tmpMin
      U     #ARY[2].CHisActive; //    AND CH2.IsActivated
      ON    #tmpMin.IsValid; //    OR NOT tmpMax.IsValid
      SPBN  mx3; // ELSE continue with CH3

      L     #ARY[2].iVAL; // THEN COPY CH2->tmpMax, because CH2 is the
      T     #tmpMax.iVAL; // act. maximum or tmpMax is not valid

      L     #ARY[2].iCH;
      T     #tmpMax.iCH;

      U     #ARY[2].CHisActive; // (if CH2 is not activated
      =     #tmpMax.IsValid; //  then tmpMax is not valid)

mx3:  L     #tmpMax.iVAL; // Channel 3 !see above documentation CH2!
      L     #ARY[3].iVAL;
      <I    ;
      U     #ARY[3].CHisActive;
      ON    #tmpMax.IsValid;
      SPBN  mx4;

      L     #ARY[3].iVAL;
      T     #tmpMax.iVAL;

      L     #ARY[3].iCH;
      T     #tmpMax.iCH;

      U     #ARY[3].CHisActive;
      =     #tmpMax.IsValid;

mx4:  L     #tmpMax.iVAL; // Channel 4
      L     #ARY[4].iVAL;
      <I    ;
      U     #ARY[4].CHisActive;
      ON    #tmpMax.IsValid;
      SPBN  mx5;

      L     #ARY[4].iVAL;
      T     #tmpMax.iVAL;

      L     #ARY[4].iCH;
      T     #tmpMax.iCH;

      U     #ARY[4].CHisActive;
      =     #tmpMax.IsValid;

mx5:  L     #tmpMax.iVAL; // If tmpMax.Val IsValid
      U     #tmpMax.IsValid;
      SPB   smax; // THEN copy the max to FC-Out

      L     0; // ELSE copy 0 to FC-Out
      T     #tmpMax.iCH;
      L     #iCH_OFF;

smax: T     #iMAX; // copy the max. to FC-Out
      L     #tmpMax.iCH; // channel no. with maximum
      T     #iNoCH_max;


END_FUNCTION

FUNCTION "m7b_Weiche_x4_INT" : VOID
TITLE =4-fach Weiche INT
//AUTOR: Stefan Maag, Dipl.-Ing. (FH) Elektrotechnik
//DATUM: 8/2018
//INTERNET: www.maagic7.de
//
//AENDERUNGSVERMERKE:
//--------------------------------------------------------------------------------
//DATUM        NAME        AENDERUNG
//--------------------------------------------------------------------------------
//15.08.2018   S.Maag      enstanden aus MUXx4xINT
//
//--------------------------------------------------------------------------------
//
//HINWEISE:
AUTHOR : 'S.Maag'
FAMILY : Maagic7
VERSION : 2.0


VAR_INPUT
  CH1 : BOOL ;
  CH2 : BOOL ;
  CH3 : BOOL ;
  CH4 : BOOL ;
  ENABLE : BOOL ;
  iValue : INT ;
END_VAR
VAR_OUTPUT
  DSP_CHANNEL : INT ;	//Displays the activated channel
END_VAR
VAR_IN_OUT
  ioINT1 : INT ;
  ioINT2 : INT ;
  ioINT3 : INT ;
  ioINT4 : INT ;
END_VAR
BEGIN
NETWORK
TITLE =

      UN    #ENABLE; // keine Freigabe, dann 0 ausgeben
      SPB   OFF;

      L     #iValue;

      U     #CH1;
      SPB   CH1;
      U     #CH2;
      SPB   CH2;
      U     #CH3;
      SPB   CH3;
      U     #CH4;
      SPB   CH4;

      SPA   OFF;

CH1:  T     #ioINT1;
      L     1; // Wert für Kanalanzeige
      SPA   SAVE;

CH2:  T     #ioINT2;
      L     2;
      SPA   SAVE;

CH3:  T     #ioINT3;
      L     3;
      SPA   SAVE;

CH4:  T     #ioINT4;
      L     4;
      SPA   SAVE;

OFF:  L     0;
      CLR   ; // EN0-Ausgang =0, da Stopp

SAVE: SAVE  ;
      T     #DSP_CHANNEL; // Anzeige aktiver Kanal

END_FUNCTION

FUNCTION "m7b_RAMP_UpDwn_INT" : VOID
TITLE =RAMP Up/Down INT
//Pro Aufruf des FC wird iUP addiert bzw. iDOWN abgezogen
//
//AUTOR: Stefan Maag, Dipl.-Ing. (FH) Elektrotechnik
//DATUM: 11/2012
//
//AENDERUNGSVERMERKE:
//--------------------------------------------------------------------------------
//DATUM        NAME      AENDERUNG
//--------------------------------------------------------------------------------
//17.04.2020   S.Maag    in Library aufgenommen
//--------------------------------------------------------------------------------
//
//HINWEISE:
AUTHOR : 'S.Maag'
FAMILY : Maagic7
VERSION : 0.1


VAR_INPUT
  iVALUE : INT ;
  iUP : INT ;
  iDOWN : INT ;
  TAKT : BOOL ;
  RESET : BOOL ;
END_VAR
VAR_IN_OUT
  memVAL : INT ;
END_VAR
BEGIN
NETWORK
TITLE =

      SET   ;
      SAVE  ;
      CLR   ;
NETWORK
TITLE =Reset

      UN    #RESET;
      SPB   ne1;
      L     #iVALUE;
      T     #memVAL;
      BEA   ;

ne1:  UN    #TAKT;
      BEB   ;

NETWORK
TITLE =Rampe maximal up/down to iValue

      L     #iVALUE;
      L     #memVAL;
      >I    ;
      SPB   up;
      <I    ;
      SPB   dwn;
      BEA   ;

up:   L     #memVAL;
      L     #iUP;
      +I    ;
      L     #iVALUE;
      >I    ;
      SPB   save;
      TAK   ;
      SPA   save;

dwn:  L     #memVAL;
      L     #iDOWN;
      -I    ;
      L     #iVALUE;
      <I    ;
      SPB   save;
      TAK   ;

save: T     #memVAL;

END_FUNCTION

FUNCTION "m7b_RP_Vortrag_INT" : VOID
TITLE =Ringpuffer Vortrag um n-Werte
//Trägt Wert in Ringpuffer von n-Werten vor. Der aktuelle Index des Puffers darf
//dabei nicht verändert werden. (ACHTUNG: Vortrag im RP ist rückwärts schreiben
//mit DEC INDEX.
//
//Dies hat den Effekt, als wäre das Produkt bereits etwas früher erfasst worden.
//Die Werte im Datenpuffer laufen dem Produkt bereits etwas voraus, was eine
//korrekte Zuordung erleichtert.
//Praktisch kombiniet man das mit freier Wegstrecke, auf dem Folgetransport.
//Unbedingt erforderlich ist der Wertevortrag, wenn z.B. mit höherer
//Geschwindigkeit auf Freilaufrollen des Folgetransports geschoben wird. Das
//Produkt würde sonst wegen der Differenzgeschwindigkeit vor den Werten herlaufen.
//Eine korrekte Zuordung der Daten wäre somit nicht möglich.
//
//iMaxLimmit begrenzt die Anzahl der vorgetragenen Werte. Somit kann man
//iNoOfValues die freie Wegstrecke nach dem Anfangssensor Transport übergeben
//und der Vortrag wird auf iMaxLimit begrenzt, falls freie Wegstrecke größer.
//
//mit iMaxLimit = iNoOfValues = 256, wird der komplette Rinpuffer mit iFillValue
//überschrieben
//
//                                              v (25=act Index)
//10 11 12 13 14 15 16 17 18 19 20 21 22 23 24 25 26 27 28 29 30 31 32 33
// 0  a  a  a  a  a  a  o  o  o  o  o  o  o  o  o
// 0  a  a  a  a  a  a  o  o  o  o  b  b  b  b  b  (Vortrag von Prod. b um 5)
//    |Vorderkante   |Hinterkante
//
//
//AUTOR: Stefan Maag, Dipl.-Ing. (FH) Elektrotechnik
//DATUM: 1/2018
//INTERNET: www.maagic7.de
//
//AENDERUNGSVERMERKE:
//--------------------------------------------------------------------------------
//DATUM        NAME        AENDERUNG
//--------------------------------------------------------------------------------
//
//--------------------------------------------------------------------------------
//
//HINWEISE:
AUTHOR : 'S.Maag'
FAMILY : Maagic7
VERSION : 0.1


VAR_INPUT
  DB_RP : BLOCK_DB ;	//Block DB: RingBuffer
  iFillValue : INT ;	//Write this value (start at act. RP_IDX)
  iNoOfValues : INT ;	//No of values to fill [0..256]
  iMaxLimit : INT ;	//Limits the NoOfValues to fill [0..256]
END_VAR
VAR_IN_OUT
  RP_IDX : INT ;	//Indexwert Ringpuffer 0..255
END_VAR
VAR_TEMP
  LoopCNT : INT ;
  tmpPTR : INT ;
END_VAR
BEGIN
NETWORK
TITLE =

      SET   ;
      SAVE  ;
      CLR   ;
NETWORK
TITLE =

      L     #RP_IDX; // actual index of Ring-Buffer
      INC   1; // INC 1 because of effective LOOP, DEC 1 will be operated first
      T     #tmpPTR;
      AUF   #DB_RP; // opens Ring-Buffer DB
NETWORK
TITLE =Min/Max Limit NoOfValues

      L     #iNoOfValues;
      L     #iMaxLimit; // MaxLimit of iNoOfValues
      >I    ;
      SPB   max;
      TAK   ; // #iNoOfValues  back to AKKU
max:  L     256; // max 256
      >I    ;
      SPB   Loop;
      TAK   ; // #iNoOfValues  back to AKKU
      L     0;
      <=I   ;
      BEB   ; // End if iNoOfValues <=0
      TAK   ; // #iNoOfValues back to AKKU
NETWORK
TITLE =LOOP to write the Values

Loop: T     #LoopCNT;
      L     #tmpPTR; // Indexwert Ringpuffer 0..255
      DEC   1;
      T     #tmpPTR; // Indexwert Ringpuffer 0..255
      SLD   4; // SLD 1 wegen DINT-Werten=>Byte + SLD 3 wegen Pointer
      L     P#0.0; // 0-Pointer addieren
      +D    ; // Pointer auf Daten erzeugen
      LAR1  ; // in Adressregister 1 laden
      L     #iFillValue; // Eingangswert laden
      T     DBW [AR1,P#0.0]; // in DB speichern
      L     #LoopCNT;
      LOOP  Loop; // Loop UP
END_FUNCTION

FUNCTION "m7b_TOL_HYS_DINT" : VOID
TITLE =Position mit Toleranzen und Hysteres prüfen [DINT]
//Anwendung:
//Toleranzprüfungen bei welchen das ok-Signal erst bei überschreiten
//einer größeren Toleranz wieder gelöscht werden soll
//
//z.B. Positionieranwendungen: nachpositionieren erst wenn Hysterseschwelle
//der Toleranz überschritten ist
//
//AUTOR: Stefan Maag, Dipl.-Ing. (FH) Elektrotechnik
//DATUM: 01/2015
//INTERNET: www.maagic7.de
//
//AENDERUNGSVERMERKE:
//--------------------------------------------------------------------------------
//DATUM        NAME        AENDERUNG
//--------------------------------------------------------------------------------
//
//--------------------------------------------------------------------------------
//
//HINWEISE:
AUTHOR : 'S.Maag'
FAMILY : Maagic7
VERSION : 0.1


VAR_INPUT
  IST : DINT ;	//Istwert Achse
  SOLL : DINT ;	//Sollwert
  TOL : DINT ;	//Toleranz Posiitionierung Achse Stop
  HYS : DINT ;	//Hysterese, Position nicht mehr o.k.
END_VAR
VAR_IN_OUT
  io_OK : BOOL ;
END_VAR
VAR_TEMP
  TOL_HYS : DINT ;
  TOL_1_OK : BOOL ;
  TOL_2_OK : BOOL ;
END_VAR
BEGIN
NETWORK
TITLE =Position mit Toleranzen und Hysterese prüfen

      L     #TOL; // Toleranz
      L     #HYS; // Hysteres
      +D    ;
      T     #TOL_HYS; // Toleranz, Hystereseschwelle

      L     #SOLL; // aktuelle Sollposition
      L     #IST; // aktuelle Istposition
      -D    ; // Positionierdifferenz
      SPP   PLUS;
      NEGD  ; // nach positiv

PLUS: L     #TOL; // Toleranz für Position ok
      <=D   ;
      S     #io_OK; // Ausgang Position ok
      TAK   ; // Positionsdifferenz in AKKU1
      L     #TOL_HYS; // Toleranz für Positionierung
      >D    ;
      R     #io_OK; // Ausgang Position ok

      U     #io_OK;
      SAVE  ;
      CLR   ;


END_FUNCTION

FUNCTION "m7b_AVG_MIN_MAX_4xDINT" : VOID
TITLE =MIN, MAX, AVERAGE from activated channels (CH1,CH2,CH3,CH4)
//Give back the minimum, maximum and average value of 4 values (channels)
//
//INPUT:
//iCH1      : value channel 1
//iCH2      : value channel 2
//iCH3      : value channel 3
//iCH4      : value channel 4
//iCH_OFF   : value is all channels are deactivated (OFF)
//
//CH1_active: FLASE: channel is deactivated (not included in calcuation)
//.           TRUE : channel is activated (included in calculation)
//.
//CH4_active:
//
//---------------------------------------------------------
//OUTPUT:
//AVG       : AVERAGE(CH1,CH2,CH3,CH4) or CH_off if all channels deactivated
//MIN       : MINIMUM(CH1,CH2,CH3,CH4) or CH_off if all channels deactivated
//MAX       : MAXIMUM(CH1,CH2,CH3,CH4) or CH_off if all channels deactivated
//NoCH_min  : Channel No. of minimum value; 0 if all channels deactivated
//NoCH_max  : Channel No. of maximum value; 0 if all channels deactivated
//NoOfActCH : Number of activated channels [0..4]
//FC-ENO    : FALSE: alle channels are disactivated; CH_OFF is selected
//            TRUE : at least 1 channel is activated; Min/Max is selected
//
//
//AUTOR: Stefan Maag, Dipl.-Ing. (FH) Elektrotechnik
//DATUM: 8/2018
//
//AENDERUNGSVERMERKE:
//--------------------------------------------------------------------------------
//DATUM        NAME      AENDERUNG
//--------------------------------------------------------------------------------
//06.08.2018   S.Maag    created by editing FC233 m7b_AVG_MIN_MAX_4xREAL
//24.09.2015   S.Maag    Function tested i.o.
//--------------------------------------------------------------------------------
//
//HINWEISE:
AUTHOR : 'S.Maag'
FAMILY : Maagic7
VERSION : 0.1


VAR_INPUT
  dCH1 : DINT ;	//Value channel 1
  dCH2 : DINT ;	//Value channel 2
  dCH3 : DINT ;	//Value channel 3
  dCH4 : DINT ;	//Value channel 4
  dCH_OFF : DINT ;	//Value if all channels are deactivated
  CH1_active : BOOL ;	//TRUE activates channel l
  CH2_active : BOOL ;	//TRUE activates channel 2
  CH3_active : BOOL ;	//TRUE activates channel 3
  CH4_active : BOOL ;	//TRUE activates channel 4
END_VAR
VAR_OUTPUT
  dAVG : DINT ;	//Average value
  dMIN : DINT ;	//Minimum value
  dMAX : DINT ;	//Maximum value
  iNoCH_min : INT ;	//Channel No of Min Value (1..3) or 0 if all channels are OFF
  iNoCH_max : INT ;	//Channel No of Max Value (1..3) or 0 if all channels are OFF
  iNoOfActCH : INT ;	//Number of activated channel [0..4]
END_VAR
VAR_TEMP
  off : BOOL ;
  tmpNoOfCHs : INT ;
  ARY : ARRAY  [1 .. 4 ] OF STRUCT
   dVAL : DINT ;
   iCH : INT ;
   CHisActive : BOOL ;
  END_STRUCT ;
  tmpMin : STRUCT
   dVAL : DINT ;
   iCH : INT ;
   IsValid : BOOL ;
  END_STRUCT ;
  tmpMax : STRUCT
   dVAL : DINT ;
   iCH : INT ;
   IsValid : BOOL ;
  END_STRUCT ;
END_VAR
BEGIN
NETWORK
TITLE =



NETWORK
TITLE =move activated channels to a temp. ARRAY & count active channels
//if a channel is not activated, it's temporary variable will be 0.0
      L     L#0; // clear temporary channel variables
      T     #ARY[1].dVAL;
      T     #ARY[2].dVAL;
      T     #ARY[3].dVAL;
      T     #ARY[4].dVAL;

      L     0; // clear the channel no.
      T     #tmpNoOfCHs;
      T     #ARY[1].iCH;
      T     #ARY[2].iCH;
      T     #ARY[3].iCH;
      T     #ARY[4].iCH;

      CLR   ;
      =     #ARY[1].CHisActive;
      =     #ARY[2].CHisActive;
      =     #ARY[3].CHisActive;
      =     #ARY[4].CHisActive;

      UN    #CH1_active; // copy CH1 if activated
      SPB   chk2;

      S     #ARY[1].CHisActive;
      L     #dCH1;
      T     #ARY[1].dVAL;
      L     1;
      T     #ARY[1].iCH;

      L     #tmpNoOfCHs;
      INC   1;
      T     #tmpNoOfCHs;

chk2: UN    #CH2_active; // copy CH2 if activated
      SPB   chk3;

      S     #ARY[2].CHisActive;
      L     #dCH2;
      T     #ARY[2].dVAL;
      L     2;
      T     #ARY[2].iCH;

      L     #tmpNoOfCHs;
      INC   1;
      T     #tmpNoOfCHs;


chk3: UN    #CH3_active; // copy CH3 if activated
      SPB   chk4;

      S     #ARY[3].CHisActive;
      L     #dCH3;
      T     #ARY[3].dVAL;
      L     3;
      T     #ARY[3].iCH;

      L     #tmpNoOfCHs;
      INC   1;
      T     #tmpNoOfCHs;


chk4: UN    #CH4_active; // copy CH4 if activated
      SPB   ne3;

      S     #ARY[4].CHisActive;
      L     #dCH4;
      T     #ARY[4].dVAL;
      L     4;
      T     #ARY[4].iCH;

      L     #tmpNoOfCHs;
      INC   1;
      T     #tmpNoOfCHs;

ne3:  NOP   0;
NETWORK
TITLE =Check: all channels OFF

      L     #tmpNoOfCHs;
      T     #iNoOfActCH; // FC Output: Number of active channels
      L     0;
      ==I   ;
      =     #off;
      NOT   ;
      SAVE  ; // ENO=FALSE if all channels are deactivated
      CLR   ;

NETWORK
TITLE =AVAERAGE (CH1, CH2, CH3, CH4)
//calculate the average of CH1..4
      L     #dCH_OFF; // if all channels are deactivated,
      U     #off; // the average value is 0.0
      SPB   sAvg; // save the avarage value

      L     #ARY[1].dVAL; // building the sum of all channels
      L     #ARY[2].dVAL; // if channel is deactivated, tmp_CH-Value is 0.0
      +D    ;
      L     #ARY[3].dVAL;
      +D    ;
      L     #ARY[4].dVAL;
      +D    ; // = CH1+CH2+CH3+CH4
      L     #tmpNoOfCHs; // number of activated channels
      /D    ;
sAvg: T     #dAVG; // the AVERAGE value of all activated channels


NETWORK
TITLE =COPY first Element of ARY to tmpMin and tmpMax
//to start min/max check with first element of CH-Array, the first Array-Element
//is copied to to the tmpMin and tmpMax structure
      L     #ARY[1].dVAL;
      T     #tmpMin.dVAL;
      T     #tmpMax.dVAL;

      L     #ARY[1].iCH;
      T     #tmpMin.iCH;
      T     #tmpMax.iCH;

      U     #ARY[1].CHisActive;
      =     #tmpMin.IsValid;
      =     #tmpMax.IsValid;

NETWORK
TITLE =Get the MINIMUM value
//
//
      L     #tmpMin.dVAL; // tempMin.Val
      L     #ARY[2].dVAL; // CH2.Val
      >D    ; // IF CH2.Val < tmpMin
      U     #ARY[2].CHisActive; //    AND CH2.IsActivated
      ON    #tmpMin.IsValid; //    OR  NOT tmpMin.IsValid
      SPBN  mn3; // ELSE continue with CH3

      L     #ARY[2].dVAL; // THEN COPY CH2->tmpMin, because CH2 is the
      T     #tmpMin.dVAL; // act. minimum or tmpMin is not valid

      L     #ARY[2].iCH;
      T     #tmpMin.iCH;

      U     #ARY[2].CHisActive; // (if CH2 is not activated
      =     #tmpMin.IsValid; //  then tmpMin is not valid)

mn3:  L     #tmpMin.dVAL; // Channel 3 !see above documentation CH2!
      L     #ARY[3].dVAL;
      >D    ;
      U     #ARY[3].CHisActive;
      ON    #tmpMin.IsValid;
      SPBN  mn4;

      L     #ARY[3].dVAL;
      T     #tmpMin.dVAL;

      L     #ARY[3].iCH;
      T     #tmpMin.iCH;

      U     #ARY[3].CHisActive;
      =     #tmpMin.IsValid;

mn4:  L     #tmpMin.dVAL; // Channel 4
      L     #ARY[4].dVAL;
      >D    ;
      U     #ARY[4].CHisActive;
      ON    #tmpMin.IsValid;
      SPBN  mn5;

      L     #ARY[4].dVAL;
      T     #tmpMin.dVAL;

      L     #ARY[4].iCH;
      T     #tmpMin.iCH;

      U     #ARY[4].CHisActive;
      =     #tmpMin.IsValid;

mn5:  L     #tmpMin.dVAL; // If tmpMin.Val IsValid
      U     #tmpMin.IsValid;
      SPB   smin; // THEN copy the min. to FC-Out

      L     0; // ELSE copy 0 to FC-Out
      T     #tmpMin.iCH;
      L     #dCH_OFF;

smin: T     #dMIN; // copy the min. to FC-Out
      L     #tmpMin.iCH; // channel no. with minimum
      T     #iNoCH_min;


NETWORK
TITLE =Get the MAXIUM value

      L     #tmpMax.dVAL; // tempMax.Val
      L     #ARY[2].dVAL; // CH2.Val
      <D    ; // IF CH2.Val > tmpMin
      U     #ARY[2].CHisActive; //    AND CH2.IsActivated
      ON    #tmpMin.IsValid; //    OR NOT tmpMax.IsValid
      SPBN  mx3; // ELSE continue with CH3

      L     #ARY[2].dVAL; // THEN COPY CH2->tmpMax, because CH2 is the
      T     #tmpMax.dVAL; // act. maximum or tmpMax is not valid

      L     #ARY[2].iCH;
      T     #tmpMax.iCH;

      U     #ARY[2].CHisActive; // (if CH2 is not activated
      =     #tmpMax.IsValid; //  then tmpMax is not valid)

mx3:  L     #tmpMax.dVAL; // Channel 3 !see above documentation CH2!
      L     #ARY[3].dVAL;
      <D    ;
      U     #ARY[3].CHisActive;
      ON    #tmpMax.IsValid;
      SPBN  mx4;

      L     #ARY[3].dVAL;
      T     #tmpMax.dVAL;

      L     #ARY[3].iCH;
      T     #tmpMax.iCH;

      U     #ARY[3].CHisActive;
      =     #tmpMax.IsValid;

mx4:  L     #tmpMax.dVAL; // Channel 4
      L     #ARY[4].dVAL;
      <D    ;
      U     #ARY[4].CHisActive;
      ON    #tmpMax.IsValid;
      SPBN  mx5;

      L     #ARY[4].dVAL;
      T     #tmpMax.dVAL;

      L     #ARY[4].iCH;
      T     #tmpMax.iCH;

      U     #ARY[4].CHisActive;
      =     #tmpMax.IsValid;

mx5:  L     #tmpMax.dVAL; // If tmpMax.Val IsValid
      U     #tmpMax.IsValid;
      SPB   smax; // THEN copy the max to FC-Out

      L     0; // ELSE copy 0 to FC-Out
      T     #tmpMax.iCH;
      L     #dCH_OFF;

smax: T     #dMAX; // copy the max. to FC-Out
      L     #tmpMax.iCH; // channel no. with maximum
      T     #iNoCH_max;


END_FUNCTION

FUNCTION "m7b_Weiche_x4_DINT" : VOID
TITLE =4-fach Weiche DINT
//AUTOR: Stefan Maag, Dipl.-Ing. (FH) Elektrotechnik
//DATUM: 8/2018
//INTERNET: www.maagic7.de
//
//AENDERUNGSVERMERKE:
//--------------------------------------------------------------------------------
//DATUM        NAME        AENDERUNG
//--------------------------------------------------------------------------------
//15.08.2018   S.Maag      enstanden aus Weiche4x_INT
//
//--------------------------------------------------------------------------------
//
//HINWEISE:
AUTHOR : 'S.Maag'
FAMILY : Maagic7
VERSION : 2.0


VAR_INPUT
  CH1 : BOOL ;
  CH2 : BOOL ;
  CH3 : BOOL ;
  CH4 : BOOL ;
  ENABLE : BOOL ;
  dValue : DINT ;
END_VAR
VAR_OUTPUT
  DSP_CHANNEL : INT ;	//Displays the activated channel
END_VAR
VAR_IN_OUT
  ioDINT1 : DINT ;
  ioDINT2 : DINT ;
  ioDINT3 : DINT ;
  ioDINT4 : DINT ;
END_VAR
BEGIN
NETWORK
TITLE =

      UN    #ENABLE; // keine Freigabe, dann 0 ausgeben
      SPB   OFF;

      L     #dValue;

      U     #CH1;
      SPB   CH1;
      U     #CH2;
      SPB   CH2;
      U     #CH3;
      SPB   CH3;
      U     #CH4;
      SPB   CH4;

      SPA   OFF;

CH1:  T     #ioDINT1;
      L     1; // Wert für Kanalanzeige
      SPA   SAVE;

CH2:  T     #ioDINT2;
      L     2;
      SPA   SAVE;

CH3:  T     #ioDINT3;
      L     3;
      SPA   SAVE;

CH4:  T     #ioDINT4;
      L     4;
      SPA   SAVE;

OFF:  L     0;
      CLR   ; // EN0-Ausgang =0, da Stopp

SAVE: SAVE  ;
      T     #DSP_CHANNEL; // Anzeige aktiver Kanal

END_FUNCTION

FUNCTION "m7b_RAMP_UpDwn_DINT" : VOID
TITLE =RAMP Up/Down INT
//Pro Aufruf des FC wird iUP addiert bzw. iDOWN abgezogen
//
//AUTOR: Stefan Maag, Dipl.-Ing. (FH) Elektrotechnik
//DATUM: 11/2012
//
//AENDERUNGSVERMERKE:
//--------------------------------------------------------------------------------
//DATUM        NAME      AENDERUNG
//--------------------------------------------------------------------------------
//17.04.2020   S.Maag    in Library aufgenommen
//--------------------------------------------------------------------------------
//
//HINWEISE:
AUTHOR : 'S.Maag'
FAMILY : Maagic7
VERSION : 0.1


VAR_INPUT
  dVALUE : DINT ;
  dUP : DINT ;
  dDOWN : DINT ;
  TAKT : BOOL ;
  RESET : BOOL ;
END_VAR
VAR_IN_OUT
  memVAL : DINT ;
END_VAR
BEGIN
NETWORK
TITLE =

      SET   ;
      SAVE  ;
      CLR   ;
NETWORK
TITLE =Reset

      UN    #RESET;
      SPB   ne1;
      L     #dVALUE;
      T     #memVAL;
      BEA   ;

ne1:  UN    #TAKT;
      BEB   ;

NETWORK
TITLE =Rampe maximal up/down to iValue

      L     #dVALUE;
      L     #memVAL;
      >D    ;
      SPB   up;
      <D    ;
      SPB   dwn;
      BEA   ;

up:   L     #memVAL;
      L     #dUP;
      +D    ;
      L     #dVALUE;
      >D    ;
      SPB   save;
      TAK   ;
      SPA   save;

dwn:  L     #memVAL;
      L     #dDOWN;
      -D    ;
      L     #dVALUE;
      <D    ;
      SPB   save;
      TAK   ;

save: T     #memVAL;

END_FUNCTION

FUNCTION "m7b_MIN_MAX_TEST_DINT" : VOID
TITLE =Test Wert auf <Min, >Max oder o.k.
//Vergleicht Wert mit Grenzen und gibt aus, wo wert liegt
//<Min, zwischen Min&Max; >Max
//
//AUTOR: Stefan Maag, Dipl.-Ing. (FH) Elektrotechnik
//DATUM: 09/2013
//
//AENDERUNGSVERMERKE:
//--------------------------------------------------------------------------------
//DATUM        NAME            AENDERUNG
//--------------------------------------------------------------------------------
//
//--------------------------------------------------------------------------------
//
//HINWEISE: 14.03.2020 in Library aufgenommen
AUTHOR : 'S.Maag'
FAMILY : Maagic7
VERSION : 0.1


VAR_INPUT
  VALUE : DINT ;	//Zu prüfender Wert
  MIN : DINT ;	//Zulässiger Minimalwert
  MAX : DINT ;	//Zulässiger Maximalwert
END_VAR
VAR_OUTPUT
  MSG_MIN : BOOL ;	//VALUE < MIN
  MSG_OK : BOOL ;	//MIN <= VALUE <= MAX
  MSG_MAX : BOOL ;	//VALUE > MAX
END_VAR
BEGIN
NETWORK
TITLE =ENO := TRUE

      SET   ;
      SAVE  ;
      CLR   ;

NETWORK
TITLE =

      L     #VALUE;
      L     #MIN;
      <R    ;
      =     #MSG_MIN;
      TAK   ;
      L     #MAX;
      >R    ;
      =     #MSG_MAX;

      UN    #MSG_MIN;
      UN    #MSG_MAX;
      =     #MSG_OK;


END_FUNCTION

FUNCTION "m7b_INTEGRATOR_REAL" : VOID
TITLE =Integrator für REAL
//TAKT: Taktgeber
//
//ENO : Zählimpuls: mit diesem Impuls den I/0-Wert 'rINTEGRAL' kopieren
//      dieser enthält zu diesem Zeitpukt den summierten Wert. Beim
//      nächsten TAKT wird dieser wieder gelöscht.
//
//AUTOR: Stefan Maag, Dipl.-Ing. (FH) Elektrotechnik
//DATUM: 09/2013
//INTERNET: www.maagic7.de
//
//AENDERUNGSVERMERKE:
//--------------------------------------------------------------------------------
//DATUM        NAME        AENDERUNG
//--------------------------------------------------------------------------------
//
//--------------------------------------------------------------------------------
//
//HINWEISE:
AUTHOR : 'S.Maag'
FAMILY : Maagic7
VERSION : 0.1


VAR_INPUT
  TAKT : BOOL ;	//Taktgeber: (Flankenauswertung erfolgt im FC)
  RESET : BOOL ;	//RESET: Zähler rücksetzen
  VALUE : REAL ;	//Zu integrierender WERT
  NoOfCounts : DINT ;	//Anzahl zu integrierender Werte
END_VAR
VAR_IN_OUT
  rINTEGRAL : REAL ;	//Integralwert
  dCOUNT : DINT ;	//Zähler
  memByte : BYTE ;	//statisches Hifls-Byte
END_VAR
VAR_TEMP
  lb0_Impuls : BOOL ;	//Lokaler Speicher:
  lb1_HM_FP_TAKT : BOOL ;	//Lokaler Speicher:
  lb2 : BOOL ;	//Lokaler Speicher:
  lb3 : BOOL ;	//Lokaler Speicher:
  lb4 : BOOL ;	//Lokaler Speicher
  lb5 : BOOL ;	//Lokaler Speicher
  lb6 : BOOL ;	//Lokaler Speicher
  lb7 : BOOL ;	//Lokaler Speicher
  tmpTAKT : BOOL ;
END_VAR
BEGIN
NETWORK
TITLE =statisches Hilfsbyte in temporäre Bits

      L     #memByte;
      T     LB     0;
      NOP   0;

NETWORK
TITLE =Impulsmerker wieder löschen, falls aktiv

      U     #lb0_Impuls;
      R     #lb0_Impuls;

NETWORK
TITLE =RESET

      UN    #RESET;
      SPB   ne4;

      L     L#0;
      T     #dCOUNT;

      L     0.000000e+000;
      T     #rINTEGRAL;

ne4:  NOP   0;
NETWORK
TITLE =Zählen

      U     #TAKT;
      FP    #lb1_HM_FP_TAKT;
      =     #tmpTAKT;

      ON    #tmpTAKT;
      O     #RESET;
      SPB   ne5;

      L     #dCOUNT; // Wenn Anzahl der Zählungen abgelaufen,
      L     #NoOfCounts; // dann Zähler rücksetzen
      <D    ;
      SPB   weit;

      L     L#0; // Zähler rücksetzten
      T     #dCOUNT;
      L     0.000000e+000;
      T     #rINTEGRAL;

weit: L     #VALUE; // Zählen
      L     #NoOfCounts;
      DTR   ;
      /R    ;
      L     #rINTEGRAL;
      +R    ;
      T     #rINTEGRAL;

      L     #dCOUNT; // Anzahl Zählungen
      +     1;
      T     #dCOUNT;

      L     #NoOfCounts; // Wenn Zählungen erreicht, dann
      >=D   ; // Impuls ausgeben
      S     #lb0_Impuls;
      SPA   ne5;

ne5:  NOP   0;

NETWORK
TITLE =FC-ENO-Ausgang = Zählimpuls

      U     #lb0_Impuls;
      SAVE  ;
      CLR   ;
NETWORK
TITLE =temporäre Bits zurück in statisches Hilfsbyte

      L     LB     0;
      T     #memByte;
      NOP   0;

END_FUNCTION

FUNCTION "m7b_IMPULS_REAL" : VOID
TITLE =Integrator mit Impuls nach Sollwert für REAL
//aufsummieren von Sensorsignalen (z.B.) kW und erzeugen eines Impulses alle
//x kWh.
//Bei z.B. einem Stromzähler der als Analogsignal die aktuelle kW-Zahl liefert,
//am besten im Takt von 1sec und NoOfCounts 3600 aufaddieren. Als Summe werden
//dann kWh geliefert. Mit rSollImpuls (z.B. 100) dann alle 100kWh einen Impuls
//ausgeben.
//
//ENO : Zählimpuls: mit diesem Impuls den I/0-Wert 'rINTEGRAL' kopieren
//      dieser enthält zu diesem Zeitpukt den summierten Wert. Beim
//      nächsten TAKT wird dieser wieder gelöscht.
//
//AUTOR: Stefan Maag, Dipl.-Ing. (FH) Elektrotechnik
//DATUM: 09/2013
//INTERNET: www.maagic7.de
//
//AENDERUNGSVERMERKE:
//--------------------------------------------------------------------------------
//DATUM        NAME        AENDERUNG
//--------------------------------------------------------------------------------
//
//--------------------------------------------------------------------------------
//
//HINWEISE:
AUTHOR : 'S.Maag'
FAMILY : Maagic7
VERSION : 0.1


VAR_INPUT
  TAKT : BOOL ;	//Taktgeber: (Flankenauswertung erfolgt im FC)
  RESET : BOOL ;	//RESET: Zähler rücksetzen
  VALUE : REAL ;	//Zu integrierender WERT
  dNoOfCounts : DINT ;	//Anzahl zu integrierender Werte
  rSollImpuls : REAL ;	//Sollwert: 1 Impuls alle 'rSollImpuls'; Sollwert bei dem 1 Impuls ausgelöst wird
END_VAR
VAR_IN_OUT
  mem_rINTEGRAL : REAL ;	//Integralwert
  memByte : BYTE ;	//statisches Hifls-Byte
END_VAR
VAR_TEMP
  lb0_Impuls : BOOL ;	//Lokaler Speicher:
  lb1_HM_FP_TAKT : BOOL ;	//Lokaler Speicher:
  lb2 : BOOL ;	//Lokaler Speicher:
  lb3 : BOOL ;	//Lokaler Speicher:
  lb4 : BOOL ;	//Lokaler Speicher
  lb5 : BOOL ;	//Lokaler Speicher
  lb6 : BOOL ;	//Lokaler Speicher
  lb7 : BOOL ;	//Lokaler Speicher
  tmpTAKT : BOOL ;
END_VAR
BEGIN
NETWORK
TITLE =statisches Hilfsbyte in temporäre Bits

      L     #memByte;
      T     LB     0;
      NOP   0;

NETWORK
TITLE =Impulsmerker wieder löschen, falls aktiv

      U     #lb0_Impuls;
      R     #lb0_Impuls;

NETWORK
TITLE =RESET

      UN    #RESET;
      SPB   ne4;

      L     0.000000e+000;
      T     #mem_rINTEGRAL;

ne4:  NOP   0;
NETWORK
TITLE =Zählen
//Bei Sollwert erreicht wird erst beim nächsten Takt der Integralwert
//zurückgesetzt, somit kann mit dem IMPULS der aktuelle Integralwert
//für die weitere Verarbeitung noch zur Verfügung gestellt werden.
//
      U     #TAKT;
      FP    #lb1_HM_FP_TAKT;
      =     #tmpTAKT;

      ON    #tmpTAKT;
      O     #RESET;
      SPB   ne5;

      L     #mem_rINTEGRAL;
      L     #rSollImpuls;
      <R    ;
      SPB   weit;

      L     #mem_rINTEGRAL; // Sollwert von Integral abziehen,
      L     #rSollImpuls; // wenn Sollwert erreicht war
      -R    ;
      T     #mem_rINTEGRAL;

weit: L     #VALUE; // Zählen
      L     #dNoOfCounts;
      DTR   ;
      /R    ;
      L     #mem_rINTEGRAL;
      +R    ;
      T     #mem_rINTEGRAL;
      L     #rSollImpuls;
      >=R   ;
      S     #lb0_Impuls; // Impuls Sollwert erreicht
      SPA   ne5;

ne5:  NOP   0;

NETWORK
TITLE =FC-ENO-Ausgang = Zählimpuls

      U     #lb0_Impuls;
      SAVE  ;
      CLR   ;
NETWORK
TITLE =temporäre Bits zurück in statisches Hilfsbyte

      L     LB     0;
      T     #memByte;
      NOP   0;

END_FUNCTION

FUNCTION "m7b_TOL_HYS_REAL" : VOID
TITLE =Position mit Toleranzen und Hysteres prüfen [REAL]
//Anwendung:
//Toleranzprüfungen bei welchen das ok-Signal erst bei überschreiten
//einer größeren Toleranz wieder gelöscht werden soll
//
//z.B. Positionieranwendungen: nachpositionieren erst wenn Hysterseschwelle
//der Toleranz überschritten ist
//
//AUTOR: Stefan Maag, Dipl.-Ing. (FH) Elektrotechnik
//DATUM: 01/2015
//INTERNET: www.maagic7.de
//
//AENDERUNGSVERMERKE:
//--------------------------------------------------------------------------------
//DATUM        NAME        AENDERUNG
//--------------------------------------------------------------------------------
//
//--------------------------------------------------------------------------------
//
//HINWEISE:
AUTHOR : 'S.Maag'
FAMILY : Maagic7
VERSION : 0.1


VAR_INPUT
  IST : DINT ;	//Istwert Achse
  SOLL : DINT ;	//Sollwert
  TOL : DINT ;	//Toleranz Posiitionierung Achse Stop
  HYS : DINT ;	//Hysterese, Position nicht mehr o.k.
END_VAR
VAR_IN_OUT
  io_OK : BOOL ;
END_VAR
VAR_TEMP
  TOL_HYS : DINT ;
  TOL_1_OK : BOOL ;
  TOL_2_OK : BOOL ;
END_VAR
BEGIN
NETWORK
TITLE =Position mit Toleranzen und Hysterese prüfen

      L     #TOL; // Toleranz
      L     #HYS; // Hysteres
      +R    ;
      T     #TOL_HYS; // Toleranz, Hystereseschwelle

      L     #SOLL; // aktuelle Sollposition
      L     #IST; // aktuelle Istposition
      -R    ; // Positionierdifferenz
      SPP   PLUS;
      NEGR  ; // nach positiv

PLUS: L     #TOL; // Toleranz für Position ok
      <=R   ;
      S     #io_OK; // Ausgang Position ok
      TAK   ; // Positionsdifferenz in AKKU1
      L     #TOL_HYS; // Toleranz für Positionierung
      >R    ;
      R     #io_OK; // Ausgang Position ok

      U     #io_OK;
      SAVE  ;
      CLR   ;


END_FUNCTION

FUNCTION "m7b_AVG_MIN_MAX_4xREAL" : VOID
TITLE =MIN, MAX, AVERAGE from activated channels (CH1,CH2,CH3,CH4)
//Give back the minimum, maximum and average value of 4 values (channels)
//
//INPUT:
//rCH1      : value channel 1
//rCH2      : value channel 2
//rCH3      : value channel 3
//rCH4      : value channel 4
//rCH_OFF   : value is all channels are deactivated (OFF)
//
//CH1_active: FLASE: channel is deactivated (not included in calcuation)
//.           TRUE : channel is activated (included in calculation)
//.
//CH4_active:
//
//---------------------------------------------------------
//OUTPUT:
//AVG       : AVERAGE(CH1,CH2,CH3,CH4) or CH_off if all channels deactivated
//MIN       : MINIMUM(CH1,CH2,CH3,CH4) or CH_off if all channels deactivated
//MAX       : MAXIMUM(CH1,CH2,CH3,CH4) or CH_off if all channels deactivated
//NoCH_min  : Channel No. of minimum value; 0 if all channels deactivated
//NoCH_max  : Channel No. of maximum value; 0 if all channels deactivated
//NoOfActCH : Number of activated channels [0..4]
//FC-ENO    : FALSE: alle channels are disactivated; CH_OFF is selected
//            TRUE : at least 1 channel is activated; Min/Max is selected
//
//
//AUTOR: Stefan Maag, Dipl.-Ing. (FH) Elektrotechnik
//DATUM: 9/2015
//
//AENDERUNGSVERMERKE:
//--------------------------------------------------------------------------------
//DATUM        NAME      AENDERUNG
//--------------------------------------------------------------------------------
//24.09.2015   S.Maag    Function tested i.o.
//--------------------------------------------------------------------------------
//
//HINWEISE:
AUTHOR : 'S.Maag'
FAMILY : Maagic7
VERSION : 0.1


VAR_INPUT
  rCH1 : REAL ;	//Value channel 1
  rCH2 : REAL ;	//Value channel 2
  rCH3 : REAL ;	//Value channel 3
  rCH4 : REAL ;	//Value channel 4
  rCH_OFF : REAL ;	//Value if all channels are deactivated
  CH1_active : BOOL ;	//TRUE activates channel l
  CH2_active : BOOL ;	//TRUE activates channel 2
  CH3_active : BOOL ;	//TRUE activates channel 3
  CH4_active : BOOL ;	//TRUE activates channel 4
END_VAR
VAR_OUTPUT
  rAVG : REAL ;	//Average value
  rMIN : REAL ;	//Minimum value
  rMAX : REAL ;	//Maximum value
  iNoCH_min : INT ;	//Channel No of Min Value (1..3) or 0 if all channels are OFF
  iNoCH_max : INT ;	//Channel No of Max Value (1..3) or 0 if all channels are OFF
  iNoOfActCH : INT ;	//Number of activated channel [0..4]
END_VAR
VAR_TEMP
  off : BOOL ;
  tmpNoOfCHs : INT ;
  ARY : ARRAY  [1 .. 4 ] OF STRUCT
   rVAL : REAL ;
   iCH : INT ;
   CHisActive : BOOL ;
  END_STRUCT ;
  tmpMin : STRUCT
   rVAL : REAL ;
   iCH : INT ;
   IsValid : BOOL ;
  END_STRUCT ;
  tmpMax : STRUCT
   rVAL : REAL ;
   iCH : INT ;
   IsValid : BOOL ;
  END_STRUCT ;
END_VAR
BEGIN
NETWORK
TITLE =



NETWORK
TITLE =move activated channels to a temp. ARRAY & count active channels
//if a channel is not activated, it's temporary variable will be 0.0
      L     0.000000e+000; // clear temporary channel variables
      T     #ARY[1].rVAL;
      T     #ARY[2].rVAL;
      T     #ARY[3].rVAL;
      T     #ARY[4].rVAL;

      L     0; // clear the channel no.
      T     #tmpNoOfCHs;
      T     #ARY[1].iCH;
      T     #ARY[2].iCH;
      T     #ARY[3].iCH;
      T     #ARY[4].iCH;

      CLR   ;
      =     #ARY[1].CHisActive;
      =     #ARY[2].CHisActive;
      =     #ARY[3].CHisActive;
      =     #ARY[4].CHisActive;

      UN    #CH1_active; // copy CH1 if activated
      SPB   chk2;

      S     #ARY[1].CHisActive;
      L     #rCH1;
      T     #ARY[1].rVAL;
      L     1;
      T     #ARY[1].iCH;

      L     #tmpNoOfCHs;
      INC   1;
      T     #tmpNoOfCHs;

chk2: UN    #CH2_active; // copy CH2 if activated
      SPB   chk3;

      S     #ARY[2].CHisActive;
      L     #rCH2;
      T     #ARY[2].rVAL;
      L     2;
      T     #ARY[2].iCH;

      L     #tmpNoOfCHs;
      INC   1;
      T     #tmpNoOfCHs;


chk3: UN    #CH3_active; // copy CH3 if activated
      SPB   chk4;

      S     #ARY[3].CHisActive;
      L     #rCH3;
      T     #ARY[3].rVAL;
      L     3;
      T     #ARY[3].iCH;

      L     #tmpNoOfCHs;
      INC   1;
      T     #tmpNoOfCHs;


chk4: UN    #CH4_active; // copy CH4 if activated
      SPB   ne3;

      S     #ARY[4].CHisActive;
      L     #rCH4;
      T     #ARY[4].rVAL;
      L     4;
      T     #ARY[4].iCH;

      L     #tmpNoOfCHs;
      INC   1;
      T     #tmpNoOfCHs;

ne3:  NOP   0;
NETWORK
TITLE =Check: all channels OFF

      L     #tmpNoOfCHs;
      T     #iNoOfActCH; // FC Output: Number of active channels
      L     0;
      ==I   ;
      =     #off;
      NOT   ;
      SAVE  ; // ENO=FALSE if all channels are deactivated
      CLR   ;

NETWORK
TITLE =AVAERAGE (CH1, CH2, CH3, CH4)
//calculate the average of CH1..4
      L     #rCH_OFF; // if all channels are deactivated,
      U     #off; // the average value is 0.0
      SPB   sAvg; // save the avarage value

      L     #ARY[1].rVAL; // building the sum of all channels
      L     #ARY[2].rVAL; // if channel is deactivated, tmp_CH-Value is 0.0
      +R    ;
      L     #ARY[3].rVAL;
      +R    ;
      L     #ARY[4].rVAL;
      +R    ; // = CH1+CH2+CH3+CH4
      L     #tmpNoOfCHs; // number of activated channels
      ITD   ;
      DTR   ;
      /R    ;
sAvg: T     #rAVG; // the AVERAGE value of all activated channels


NETWORK
TITLE =COPY first Element of ARY to tmpMin and tmpMax
//to start min/max check with first element of CH-Array, the first Array-Element
//is copied to to the tmpMin and tmpMax structure
      L     #ARY[1].rVAL;
      T     #tmpMin.rVAL;
      T     #tmpMax.rVAL;

      L     #ARY[1].iCH;
      T     #tmpMin.iCH;
      T     #tmpMax.iCH;

      U     #ARY[1].CHisActive;
      =     #tmpMin.IsValid;
      =     #tmpMax.IsValid;

NETWORK
TITLE =Get the MINIMUM value
//
//
      L     #tmpMin.rVAL; // tempMin.Val
      L     #ARY[2].rVAL; // CH2.Val
      >R    ; // IF CH2.Val < tmpMin
      U     #ARY[2].CHisActive; //    AND CH2.IsActivated
      ON    #tmpMin.IsValid; //    OR  NOT tmpMin.IsValid
      SPBN  mn3; // ELSE continue with CH3

      L     #ARY[2].rVAL; // THEN COPY CH2->tmpMin, because CH2 is the
      T     #tmpMin.rVAL; // act. minimum or tmpMin is not valid

      L     #ARY[2].iCH;
      T     #tmpMin.iCH;

      U     #ARY[2].CHisActive; // (if CH2 is not activated
      =     #tmpMin.IsValid; //  then tmpMin is not valid)

mn3:  L     #tmpMin.rVAL; // Channel 3 !see above documentation CH2!
      L     #ARY[3].rVAL;
      >R    ;
      U     #ARY[3].CHisActive;
      ON    #tmpMin.IsValid;
      SPBN  mn4;

      L     #ARY[3].rVAL;
      T     #tmpMin.rVAL;

      L     #ARY[3].iCH;
      T     #tmpMin.iCH;

      U     #ARY[3].CHisActive;
      =     #tmpMin.IsValid;

mn4:  L     #tmpMin.rVAL; // Channel 4
      L     #ARY[4].rVAL;
      >R    ;
      U     #ARY[4].CHisActive;
      ON    #tmpMin.IsValid;
      SPBN  mn5;

      L     #ARY[4].rVAL;
      T     #tmpMin.rVAL;

      L     #ARY[4].iCH;
      T     #tmpMin.iCH;

      U     #ARY[4].CHisActive;
      =     #tmpMin.IsValid;

mn5:  L     #tmpMin.rVAL; // If tmpMin.Val IsValid
      U     #tmpMin.IsValid;
      SPB   smin; // THEN copy the min. to FC-Out

      L     0; // ELSE copy 0 to FC-Out
      T     #tmpMin.iCH;
      L     #rCH_OFF;

smin: T     #rMIN; // copy the min. to FC-Out
      L     #tmpMin.iCH; // channel no. with minimum
      T     #iNoCH_min;


NETWORK
TITLE =Get the MAXIUM value

      L     #tmpMax.rVAL; // tempMax.Val
      L     #ARY[2].rVAL; // CH2.Val
      <R    ; // IF CH2.Val > tmpMin
      U     #ARY[2].CHisActive; //    AND CH2.IsActivated
      ON    #tmpMin.IsValid; //    OR NOT tmpMax.IsValid
      SPBN  mx3; // ELSE continue with CH3

      L     #ARY[2].rVAL; // THEN COPY CH2->tmpMax, because CH2 is the
      T     #tmpMax.rVAL; // act. maximum or tmpMax is not valid

      L     #ARY[2].iCH;
      T     #tmpMax.iCH;

      U     #ARY[2].CHisActive; // (if CH2 is not activated
      =     #tmpMax.IsValid; //  then tmpMax is not valid)

mx3:  L     #tmpMax.rVAL; // Channel 3 !see above documentation CH2!
      L     #ARY[3].rVAL;
      <R    ;
      U     #ARY[3].CHisActive;
      ON    #tmpMax.IsValid;
      SPBN  mx4;

      L     #ARY[3].rVAL;
      T     #tmpMax.rVAL;

      L     #ARY[3].iCH;
      T     #tmpMax.iCH;

      U     #ARY[3].CHisActive;
      =     #tmpMax.IsValid;

mx4:  L     #tmpMax.rVAL; // Channel 4
      L     #ARY[4].rVAL;
      <R    ;
      U     #ARY[4].CHisActive;
      ON    #tmpMax.IsValid;
      SPBN  mx5;

      L     #ARY[4].rVAL;
      T     #tmpMax.rVAL;

      L     #ARY[4].iCH;
      T     #tmpMax.iCH;

      U     #ARY[4].CHisActive;
      =     #tmpMax.IsValid;

mx5:  L     #tmpMax.rVAL; // If tmpMax.Val IsValid
      U     #tmpMax.IsValid;
      SPB   smax; // THEN copy the max to FC-Out

      L     0; // ELSE copy 0 to FC-Out
      T     #tmpMax.iCH;
      L     #rCH_OFF;

smax: T     #rMAX; // copy the max. to FC-Out
      L     #tmpMax.iCH; // channel no. with maximum
      T     #iNoCH_max;


END_FUNCTION

FUNCTION "m7b_Weiche_x4_REAL" : VOID
TITLE =4-fach Weiche REAL
//AUTOR: Stefan Maag, Dipl.-Ing. (FH) Elektrotechnik
//DATUM: 8/2018
//INTERNET: www.maagic7.de
//
//AENDERUNGSVERMERKE:
//--------------------------------------------------------------------------------
//DATUM        NAME        AENDERUNG
//--------------------------------------------------------------------------------
//15.08.2018   S.Maag      enstanden aus Weiche4x_INT
//
//--------------------------------------------------------------------------------
//
//HINWEISE:
AUTHOR : 'S.Maag'
FAMILY : Maagic7
VERSION : 2.0


VAR_INPUT
  CH1 : BOOL ;
  CH2 : BOOL ;
  CH3 : BOOL ;
  CH4 : BOOL ;
  ENABLE : BOOL ;
  rValue : DINT ;
END_VAR
VAR_OUTPUT
  DSP_CHANNEL : INT ;	//Displays the activated channel
END_VAR
VAR_IN_OUT
  ioREAL1 : REAL ;
  ioREAL2 : REAL ;
  ioREAL3 : REAL ;
  ioREAL4 : REAL ;
END_VAR
BEGIN
NETWORK
TITLE =

      UN    #ENABLE; // keine Freigabe, dann 0 ausgeben
      SPB   OFF;

      L     #rValue;

      U     #CH1;
      SPB   CH1;
      U     #CH2;
      SPB   CH2;
      U     #CH3;
      SPB   CH3;
      U     #CH4;
      SPB   CH4;

      SPA   OFF;

CH1:  T     #ioREAL1;
      L     1; // Wert für Kanalanzeige
      SPA   SAVE;

CH2:  T     #ioREAL2;
      L     2;
      SPA   SAVE;

CH3:  T     #ioREAL3;
      L     3;
      SPA   SAVE;

CH4:  T     #ioREAL4;
      L     4;
      SPA   SAVE;

OFF:  L     0;
      CLR   ; // EN0-Ausgang =0, da Stopp

SAVE: SAVE  ;
      T     #DSP_CHANNEL; // Anzeige aktiver Kanal

END_FUNCTION

FUNCTION "m7b_RAMP_UpDwn_REAL" : VOID
TITLE =RAMP Up/Down REAL
//Pro Aufruf des FC wird rUP addiert bzw. rDOWN abgezogen
//
//AUTOR: Stefan Maag, Dipl.-Ing. (FH) Elektrotechnik
//DATUM: 11/2012
//
//AENDERUNGSVERMERKE:
//--------------------------------------------------------------------------------
//DATUM        NAME      AENDERUNG
//--------------------------------------------------------------------------------
//17.04.2020   S.Maag    in Library aufgenommen
//--------------------------------------------------------------------------------
//
//HINWEISE:
AUTHOR : 'S.Maag'
FAMILY : Maagic7
VERSION : 0.1


VAR_INPUT
  rVALUE : REAL ;
  rUP : REAL ;
  rDOWN : REAL ;
  TAKT : BOOL ;
  RESET : BOOL ;
END_VAR
VAR_IN_OUT
  memVAL : REAL ;
END_VAR
BEGIN
NETWORK
TITLE =

      SET   ;
      SAVE  ;
      CLR   ;
NETWORK
TITLE =Reset

      UN    #RESET;
      SPB   ne1;
      L     #rVALUE;
      T     #memVAL;
      BEA   ;

ne1:  UN    #TAKT;
      BEB   ;

NETWORK
TITLE =Rampe maximal up/down to rValue

      L     #rVALUE;
      L     #memVAL;
      >R    ;
      SPB   up;
      <R    ;
      SPB   dwn;
      BEA   ;

up:   L     #memVAL;
      L     #rUP;
      +R    ;
      L     #rVALUE;
      >R    ;
      SPB   save;
      TAK   ;
      SPA   save;

dwn:  L     #memVAL;
      L     #rDOWN;
      -R    ;
      L     #rVALUE;
      <R    ;
      SPB   save;
      TAK   ;

save: T     #memVAL;

END_FUNCTION

FUNCTION "m7b_RoundReal" : REAL
TITLE =Round a REAL to No of digits / Runden auf Anzahl Kommastellen
//AUTOR: Stefan Maag, Dipl.-Ing. (FH) Elektrotechnik
//DATUM: 3/2017
//INTERNET: www.maagic7.de
//
//AENDERUNGSVERMERKE:
//--------------------------------------------------------------------------------
//DATUM        NAME        AENDERUNG
//--------------------------------------------------------------------------------
//
//--------------------------------------------------------------------------------
//
//HINWEISE:
AUTHOR : 'S.Maag'
FAMILY : Maagic7
VERSION : 0.1


VAR_INPUT
  rIN : REAL ;	//REAL Value to round
  iNoOfDigits : INT ;	//No of digits after the dot / Nachkommastellen
END_VAR
BEGIN
NETWORK
TITLE =
//How to round a REAL to No of digits after the komma.
//
//ROUNDED_REAL = DINT_TO_REAL (REAL_TO_DINT (IN_REAL * Factor)) / Factor
//Factor for 1 digit = 10, for 2 digits = 100 ...
//
//1. Create a factor from No of digits
//
//   Digits  Factor
//      0             1
//      1            10
//      2           100
//      3         1.000
//      4        10.000
//      5       100.000  This is the possible maximum
//                       because S7-REAL has 6 digits max.
//
//   We start with creating the factor as BCD No, so we have to shift left
//   the BCD No '1' iNoOfDigits
//   Each BCD No has 4 Btis, so we have to Shift Bits := iNoOfDigits * 4
//
//      L     #iNoOfDigits                // No. of digits after komma
//      SLW   2                           // *4 Bits per BCD No.
//      L     1                           // Load a BCD 1 to Akku
//      SLD
//
//After this we get a BCD No:  1/10/100/1000 ...
//
//Wit BTD we convert this to a INT, with DTR to our REAL Factor for digits
//
//2. We cut unneeded digits
//   IN_REAL * Factor
//   REAL_TO_DINT        // cut the unneeded digits
//   DINT_TO_REAL        // back to REAL
//   / Factor
//   = Rounded REAL
      L     #iNoOfDigits; // No. of digits after komma
      L     5; // maximum of possible digits
      >I    ;
      SPB   err; // If iNoOfDigits >5 THEN err
      TAK   ;
      L     0; // If iNoOfDigits <0 THEN err
      <I    ;
      SPB   err;
      SPA   do;

err:  L     #rIN; // IF err THEN  RET_VAL = rIN
      SPA   save;

do:   L     #iNoOfDigits; // No. of digits after komma
      SLW   2; // *4 Bits per BCD No.
      L     1; // Load a BCD 1 to Akku
      SLD   ; // Shift the BCD '1' No of digits left
      BTD   ; // convert the BCD 1/10/100/1000 ... to INT := 10 EXP iKomma
      DTR   ; // convert Factor  1/10/100/1000 to REAL
      PUSH  ; // Fill AKKU 2/3 with Factor
      PUSH  ; // it's because of automatic POP at 4 Akku CPU's
      L     #rIN; // Load the IN_REAL VALUE
      *R    ; // = IN_REAL * DigitFactor (1/10/100/1000 ...)
      RND   ; // Round to DINT
      DTR   ; // DINT_TO_REAL (=> without komma)
      TAK   ; // Factor back to AKKU 1, Rounded (Value*Factor) to AKKU 2
      /R    ; // = (RoundedValue * Factor) / Factor
save: T     #RET_VAL; // Result rounded to no of digits after komma

      SET   ;
      SAVE  ;


END_FUNCTION

FUNCTION "m7b_MinMax_2xREAL" : REAL
TITLE =Select min. or. max of 2 REAL values
//Select the minimum or maximum of 2 REAL values.
//
//INPUT:
//rCH1      : value channel 1
//rCH2      : value channel 2
//cfgMinMax : FALSE: select the min: MIN(CH1,CH2)
//            TRUE : select the max: MAX(CH1,CH2)
//---------------------------------------------------------
//OUTPUT:
//RET_VAL   : the selected value min or max., depending on cfgMinMax
//ENO       : FALSE = CH1 is selected
//            TRUE  = CH2 is selected
//
//AUTOR: Stefan Maag, Dipl.-Ing. (FH) Elektrotechnik
//DATUM: 09/2015
//INTERNET: www.maagic7.de
//
//AENDERUNGSVERMERKE:
//--------------------------------------------------------------------------------
//DATUM        NAME            AENDERUNG
//--------------------------------------------------------------------------------
//
//--------------------------------------------------------------------------------
//
//HINWEISE:
AUTHOR : 'S.Maag'
FAMILY : Maagic7
VERSION : 0.1


VAR_INPUT
  rCH1 : REAL ;	//Value channel 1
  rCH2 : REAL ;	//Value channel 2
  cfgMinMax : BOOL ;	//FALSE: select min. value; TRUE: select max. Value
END_VAR
BEGIN
NETWORK
TITLE =

      U     #cfgMinMax;
      SPB   MAX;
      SPA   MIN;

NETWORK
TITLE =Select max (greater vlaue)

MAX:  L     #rCH1;
      L     #rCH2;
      <R    ; // TRUE if CH1<CH2 := CH2 is max
      SAVE  ; // ENO (BIE) = TRUE if CH2 selected
      SPB   SAVE;
      TAK   ;
      SPA   SAVE;

NETWORK
TITLE =Select min (lower vlaue)

MIN:  L     #rCH1;
      L     #rCH2;
      >R    ; // TRUE if CH1>CH2 := CH2 is min
      SAVE  ; // ENO (BIE) = TRUE if CH2 selected
      SPB   SAVE;
      TAK   ;
      SPA   SAVE;

NETWORK
TITLE =

SAVE: T     #RET_VAL; // Return the selected value

END_FUNCTION

FUNCTION "m7b_MIN_MAX_TEST_REAL" : VOID
TITLE =Test Wert auf <Min, >Max oder o.k.
//Vergleicht Wert mit Grenzen und gibt aus, wo wert liegt
//<Min, zwischen Min&Max; >Max
//
//AUTOR: Stefan Maag, Dipl.-Ing. (FH) Elektrotechnik
//DATUM: 09/2013
//INTERNET: www.maagic7.de
//
//AENDERUNGSVERMERKE:
//--------------------------------------------------------------------------------
//DATUM        NAME            AENDERUNG
//--------------------------------------------------------------------------------
//
//--------------------------------------------------------------------------------
//
//HINWEISE:
AUTHOR : 'S.Maag'
FAMILY : Maagic7
VERSION : 0.1


VAR_INPUT
  VALUE : REAL ;	//Zu prüfender Wert
  MIN : REAL ;	//Zulässiger Minimalwert
  MAX : REAL ;	//Zulässiger Maximalwert
END_VAR
VAR_OUTPUT
  MSG_MIN : BOOL ;	//VALUE < MIN
  MSG_OK : BOOL ;	//MIN <= VALUE <= MAX
  MSG_MAX : BOOL ;	//VALUE > MAX
END_VAR
BEGIN
NETWORK
TITLE =ENO := TRUE

      SET   ;
      SAVE  ;
      CLR   ;

NETWORK
TITLE =

      L     #VALUE;
      L     #MIN;
      <R    ;
      =     #MSG_MIN;
      TAK   ;
      L     #MAX;
      >R    ;
      =     #MSG_MAX;

      UN    #MSG_MIN;
      UN    #MSG_MAX;
      =     #MSG_OK;


END_FUNCTION

FUNCTION "m7b_DampingReal" : VOID
TITLE =Damping of a REAL value
//AUTOR: Stefan Maag, Dipl.-Ing. (FH) Elektrotechnik
//DATUM: 9/2015
//INTERNET: www.maagic7.de
//
//AENDERUNGSVERMERKE:
//--------------------------------------------------------------------------------
//DATUM        NAME            AENDERUNG
//--------------------------------------------------------------------------------
//28.11.2017   S.Maag        Fehlerabragen SPU err hinzugefügt, da es
//                           bei ungültigen Gleitpunktzahlen zu einem
//                           Dauerhaften Fehler kommt, der sich selbst nicht
//                           mehr korrigiert, da die Rechnung abgebrochen wird.
//                           Das ist ein sehr seltens Phänomen und konnte nicht
//                           ganz nachvollzogen werden warum das passiert.
//                           in der Gleitpunktzahl steht dann der HEX-WERT
//                           DW#16#7FC0 0000
//                           Aufgetaucht ist dies nach einem Sensordefekt und
//                           Sensorwechsel (Wiegezelle)
//--------------------------------------------------------------------------------
//
//HINWEISE:
AUTHOR : 'S.Maag'
FAMILY : Maagic7
VERSION : 0.1


VAR_INPUT
  rVALUE : REAL ;
  rising_edge_1s : BOOL ;
  rDampingFactor : REAL ;
END_VAR
VAR_IN_OUT
  IO_VALUE_DAMP : REAL ;
END_VAR
VAR_TEMP
  rDamping : REAL ;
END_VAR
BEGIN
NETWORK
TITLE =



NETWORK
TITLE =Dämpfung des Sensorwertes
//Durch das aufaddieren eines Teils der Differenz zum aktuellen Analogwert
//läuft der gedämpfte Wert dem Analogwert immer etwas hinterher. Es ergibt sich
//ein exponentieller Nachlauf (vgl. Kondensator Ladekurve) bei einem
//Dämpfungsfaktor von 2 erhält man nach 5 Impulsen ca. 96.9%, nach 7 Impulsen ca.
//99.2% Sensorwertes. Je höher der Dämpfungsfaktor, desto langsamer läuft der
//Wert hinterher.
//
      UN    #rising_edge_1s;
      SPB   ne6;

      L     #rDampingFactor; // sicherstellen, dass
      L     1.000000e+000; // Dämpfungsfaktor >=1.0
      <R    ;
      SPB   sav;
      TAK   ;
sav:  T     #rDamping;

      L     #rVALUE;
      L     #IO_VALUE_DAMP;
      -R    ;
      SPU   err; // Wenn Fehler, z.B. ungültige Gleitpunktzahl
      L     #rDamping;
      /R    ;
      SPU   err; // Wenn Fehler, z.B. ungültige Gleitpunktzahl
      L     #IO_VALUE_DAMP;
      +R    ;
      SPU   err; // Wenn Fehler, z.B. ungültige Gleitpunktzahl
      T     #IO_VALUE_DAMP;
      BEA   ;

err:  L     #rVALUE; // Wenn Fehler, dann Eingangswert direkt
      T     #IO_VALUE_DAMP; // durchschleusen
ne6:  NOP   0;
END_FUNCTION

FUNCTION "m7b_PE_to_DB" : VOID
TITLE =PE_to_DB: kopiert einen Peripherie Eingangsbereich in DB
//Kopiert eine Anzahl von Bytes PE zu DB. Die Kopierroutine arbeitet sehr
//effektiv, da die Werte nicht als einzelne Bytes sondern
//als 32-Bit-Werte kopiert werden.
//
//AUTOR: Stefan Maag, Dipl.-Ing. (FH) Elektrotechnik
//DATUM: 11/2011
//INTERNET: www.maagic7.de
//
//AENDERUNGSVERMERKE:
//--------------------------------------------------------------------------------
//DATUM        NAME        AENDERUNG
//--------------------------------------------------------------------------------
//
//--------------------------------------------------------------------------------
//
//HINWEISE:
AUTHOR : 'S.Maag'
FAMILY : Maagic7
VERSION : 0.1


VAR_INPUT
  ADR_PE : INT ;	//Start Adresse Peripherie Eingangsbereich
  DB_NR : BLOCK_DB ;	//DB
  DB_ADR : INT ;	//Byteadresse im DB
  BYTES : INT ;	//Number of Bytes to copy
END_VAR
VAR_TEMP
  QUELL_ADR : DINT ;
  ZIEL_ADR : DINT ;
  AR1 : DINT ;
  AR2 : DINT ;
END_VAR
BEGIN
NETWORK
TITLE =Register sichern

      SET   ;
      SAVE  ;
      CLR   ;

NETWORK
TITLE =Register sichern

      TAR1  #AR1; // Adressregister 1 sichern
      TAR2  #AR2; // Adressregister 2 sichern

NETWORK
TITLE =Adressen für Quell und Ziel-DW als Pointer in Adressregister

      L     #ADR_PE; // Quelladresse-PE
      SLD   3; // als Pointer
      L     P#0.0; // 0-Pointer addieren, damit
      +D    ; // Kennungsbits für Pointer gesetzt werden
      LAR1  ; // ins Adressregister 1

      L     #DB_ADR; // Zieldatenwort-Nr
      SLD   3; // als Pointer
      L     P#0.0;
      +D    ;
      LAR2  ; // ins Adressregister 2
NETWORK
TITLE =Daten kopieren

      AUF   #DB_NR; // Ziel-DB als Global-DB öffnen

      L     #BYTES; // Anzahl der zu kopierenden Bytes
      SRW   2; // in Anzahl der 32-Bit-Werte umrechen
LOOP: L     PED [AR1,P#0.0]; // Quell: PED lesen
      T     DBD [AR2,P#0.0]; // Ziel-Daten schreiben
      +AR1  P#4.0; // Quell-Pointer in AR1 um 4 Bytes erhöhen
      +AR2  P#4.0; // Ziel-Pointer in AR2 um 4 Bytes erhöhen
      TAK   ; // Schleifenzähler wieder in Akku 1 zurück
      LOOP  LOOP; // Schleifenzähler bearbeiten

      L     #BYTES; // nun noch prüfen ob noch ein 16-Bit-Wert kopiert werden muss
      SRW   2; // LSB von Anzahl wird in Ergebnisvorzeichenregister geschoben
      SPZ   BYT; // prüft somit, ob LSB von ANZAHL = 1 ist
      L     PEW [AR1,P#0.0]; // Dann muss das letze DW noch kopiert werden
      T     DBW [AR2,P#0.0];
      +AR1  P#2.0; // Quell-Pointer in AR1 um 4 Bytes erhöhen
      +AR2  P#2.0; // Ziel-Pointer in AR2 um 4 Bytes erhöhen

BYT:  L     #BYTES; // nun noch prüfen ob noch ein 8-Bit-Wert kopiert werden muss
      SRW   1; // LSB von Anzahl wird in Ergebnisvorzeichenregister geschoben
      SPZ   END; // prüft somit, ob LSB von ANZAHL = 1 ist
      L     PEB [AR1,P#0.0]; // Dann muss das letze Byte noch kopiert werden
      T     DBB [AR2,P#0.0];
END:  NOP   0;

NETWORK
TITLE =Registerinhalte wieder herstellen

      LAR1  #AR1; // Adressregister 1 wieder herstellen
      LAR2  #AR2; // Adressregister 2 wieder herstellen
END_FUNCTION

FUNCTION "m7b_DB_to_PA" : VOID
TITLE =DB_to_PA: kopiert Daten von einem DB zu PeripherieAusgängen
//Kopiert eine Anzahl von Bytes von DB zu PA
//Die Kopierroutine arbeitet sehr effektiv, da die Werte nicht als einzelne Bytes
//sondern als 32-Bit-Werte kopiert werden.
//
//AUTOR: Stefan Maag, Dipl.-Ing. (FH) Elektrotechnik
//DATUM: 11/2011
//INTERNET: www.maagic7.de
//
//AENDERUNGSVERMERKE:
//--------------------------------------------------------------------------------
//DATUM        NAME        AENDERUNG
//--------------------------------------------------------------------------------
//
//--------------------------------------------------------------------------------
//
//HINWEISE:
AUTHOR : 'S.Maag'
FAMILY : Maagic7
VERSION : 0.1


VAR_INPUT
  ADR_PA : INT ;	//Anfangs-Adresse Peripherie Ausgangsblock
  DB_Nr : BLOCK_DB ;	//DB
  DB_ADR : INT ;	//Byte Adresse im DB
  BYTES : INT ;	//Number of bytes
END_VAR
VAR_TEMP
  QUELL_ADR : DINT ;
  ZIEL_ADR : DINT ;
  AR1 : DINT ;
  AR2 : DINT ;
END_VAR
BEGIN
NETWORK
TITLE =Register sichern

      SET   ;
      SAVE  ;
      CLR   ;

NETWORK
TITLE =Register sichern

      TAR1  #AR1; // Adressregister 1 sichern
      TAR2  #AR2; // Adressregister 2 sichern

NETWORK
TITLE =Adressen für Quelle und Ziel als Pointer in Adressregister

      L     #DB_ADR; // Quelladresse Datenwort-Nr
      SLD   3; // als Pointer
      L     P#0.0;
      +D    ;
      LAR1  ; // ins Adressregister 1

      L     #ADR_PA; // Zieladresse PA
      SLD   3; // als Pointer
      L     P#0.0; // 0-Pointer addieren, damit
      +D    ; // Kennungsbits für Pointer gesetzt werden
      LAR2  ; // ins Adressregister 2
NETWORK
TITLE =Daten kopieren

      AUF   #DB_Nr; // Ziel-DB als Global-DB öffnen

      L     #BYTES; // Anzahl der zu kopierenden Bytes
      SRW   2; // in Anzahl der 32-Bit-Werte umrechen
LOOP: L     DBD [AR1,P#0.0]; // Quell: DBD lesen
      T     PAD [AR2,P#0.0]; // Ziel PAD speichern
      +AR1  P#4.0; // Quell-Pointer in AR1 um 4 Bytes erhöhen
      +AR2  P#4.0; // Ziel-Pointer in AR2 um 4 Bytes erhöhen
      TAK   ; // Schleifenzähler wieder in Akku 1 zurück
      LOOP  LOOP; // Schleifenzähler bearbeiten

      L     #BYTES; // nun noch prüfen ob noch ein 16-Bit-Wert kopiert werden muss
      SRW   2; // LSB von Anzahl wird in Ergebnisvorzeichenregister geschoben
      SPZ   BYT; // prüft somit, ob LSB von ANZAHL = 1 ist
      L     DBW [AR1,P#0.0]; // Dann muss das letze DW noch kopiert werden
      T     PAW [AR2,P#0.0];
      +AR1  P#2.0; // Quell-Pointer in AR1 um 4 Bytes erhöhen
      +AR2  P#2.0; // Ziel-Pointer in AR2 um 4 Bytes erhöhen

BYT:  L     #BYTES; // nun noch prüfen ob noch ein 8-Bit-Wert kopiert werden muss
      SRW   1; // LSB von Anzahl wird in Ergebnisvorzeichenregister geschoben
      SPZ   END; // prüft somit, ob LSB von ANZAHL = 1 ist
      L     DBB [AR1,P#0.0]; // Dann muss das letze Byte noch kopiert werden
      T     PAB [AR2,P#0.0];
END:  NOP   0;

NETWORK
TITLE =Registerinhalte wieder herstellen

      LAR1  #AR1; // Adressregister 1 wieder herstellen
      LAR2  #AR2; // Adressregister 2 wieder herstellen
END_FUNCTION

FUNCTION "m7b_BitToANY" : ANY
TITLE =BitToANY: 2x ANY Multiplexer
//AUTOR: Stefan Maag, Dipl.-Ing. (FH) Elektrotechnik
//DATUM: 10/2008
//INTERNET: www.maagic7.de
//
//AENDERUNGSVERMERKE:
//--------------------------------------------------------------------------------
//DATUM        NAME        AENDERUNG
//--------------------------------------------------------------------------------
//01.04.2020   S.Maag      von 2xAnyMultiPlexer nach BitToANY umbenannt, da
//                         kein echter Multiplexer, sondern ähnlich wie
//                         die Funktionen BitToDINT, BitToReal, eine
//                         Einfachauswahl. Dazu ebenfalls die Auswahleingänge
//                         S1/S2 gegen nur einen Eingang BIT ersetzt.
//                         D.h. es gibt nur eine Entweder Oder Auswahl.
//                         Grund: Würde bei S1/S2 nichts ausgewählt, dann
//                         würden willkührliche Daten als RET_VAL zurückgegeben.
//                         Beim 3x/4xAnyMultiplexer wurde dies mit eiem temp.
//                         NullAny behoben. Bei 2-fach macht das aber keinen
//                         Sinn. Hier ist die bessere Lösung eine Muss-Auswahl.
//--------------------------------------------------------------------------------
//
//HINWEISE:
AUTHOR : 'S.Maag'
FAMILY : Maagic7
VERSION : 0.1


VAR_INPUT
  BIT : BOOL ;
  ANY0 : ANY ;	//ANY Pointer 0
  ANY1 : ANY ;	//ANY Pointer 1
END_VAR
BEGIN
NETWORK
TITLE =
//It isn't recomended to restore AR2, it will be done automatically by the
//systems CALL operation, when leaving the Function
      U     #BIT; // Select No. 1
      SAVE  ;
      SPB   HIGH;
      L     P##ANY0; // Load the Pointer of ANY 0
      SPA   SAVE;
HIGH: L     P##ANY1; // Load the Pointer of ANY 1
SAVE: LAR1  ; // Load the Pointer of the Source Any into AR1
      L     P##RET_VAL; // Load the Pointer of the ReturnValue into
      LAR2  ; // AR2

      L     D [AR1,P#0.0]; // Copy the 10 Bytes of the ANY Pointer to
      T     D [AR2,P#0.0]; // the returned ANY

      L     D [AR1,P#4.0];
      T     D [AR2,P#4.0];

      L     W [AR1,P#8.0];
      T     W [AR2,P#8.0];


END_FUNCTION

FUNCTION "m7b_MUXx3xANY" : ANY
TITLE =3x ANY Multiplexer
//AUTOR: Stefan Maag, Dipl.-Ing. (FH) Elektrotechnik
//DATUM: 10/2008
//INTERNET: www.maagic7.de
//
//AENDERUNGSVERMERKE:
//--------------------------------------------------------------------------------
//DATUM        NAME        AENDERUNG
//--------------------------------------------------------------------------------
//01.04.2020   S.Maag      Anzeige aktiver Kanal (DSP_CHANNEL)
//                         RETURN NullAny, wenn kein Kanal ausgewählt
//                         ENABLE wie bei WerteMultiplexern hinzugefügt
//--------------------------------------------------------------------------------
//
//HINWEISE:
AUTHOR : 'S.Maag'
FAMILY : Maagic7
VERSION : 0.1


VAR_INPUT
  S1 : BOOL ;	//Select no. 1
  S2 : BOOL ;	//Select no. 2
  S3 : BOOL ;	//Select no. 3
  ENABLE : BOOL ;	//If not Enabled: RET_VAL:=NullAny
  ANY1 : ANY ;	//ANY Pointer 1
  ANY2 : ANY ;	//ANY Pointer 3
  ANY3 : ANY ;	//ANY Pointer 3
END_VAR
VAR_OUTPUT
  DSP_CHANNEL : INT ;	//Displays the activated channel
END_VAR
VAR_TEMP
  anyNull : ANY ;
END_VAR
BEGIN
NETWORK
TITLE =
//It isn't recomended to restore AR1 & AR2, it will be done automatically by the
//systems CALL operation, when leaving the Function
      UN    #ENABLE; // keine Freigabe, dann 0 ausgeben
      SPB   OFF;

      U     #S1; // Select No. 1
      SPB   S1;
      U     #S2; // Select No. 2
      SPB   S2;
      U     #S3; // Select No. 3
      SPB   S3;
      SPA   OFF;

S1:   L     P##ANY1; // Load the Pointer of ANY 1
      L     1; // Wert für Kanalanzeige
      SPA   SAVE;
S2:   L     P##ANY2; // Load the Pointer of ANY 2
      L     2;
      SPA   SAVE;
S3:   L     P##ANY3; // Load the Pointer of ANY 3
      L     3;
      SPA   SAVE;

OFF:  L     P##anyNull; // Create a temporary
      LAR1  ; // NullAny
      L     DW#16#0;
      T     D [AR1,P#0.0];
      T     D [AR1,P#4.0];
      T     W [AR1,P#8.0];

      L     P##anyNull; // Load Pointer to temporary NullAny
      L     0;
      CLR   ; // CLR BIE

SAVE: SAVE  ; // FC-ENO: TRUE IF ChannelSelected
      T     #DSP_CHANNEL; // Anzeige aktiver Kanal
      TAK   ; // P##ANY in AKKU1 zurück
      LAR1  ; // Load the Pointer of the Source Any into AR1
      L     P##RET_VAL; // Load the Pointer of the ReturnValue into
      LAR2  ; // AR2

      L     D [AR1,P#0.0]; // Copy the 10 Bytes of the ANY Pointer to
      T     D [AR2,P#0.0]; // the returned ANY

      L     D [AR1,P#4.0];
      T     D [AR2,P#4.0];

      L     W [AR1,P#8.0];
      T     W [AR2,P#8.0];


END_FUNCTION

FUNCTION "m7b_MUXx4xANY" : ANY
TITLE =4x ANY Multiplexer
//AUTOR: Stefan Maag, Dipl.-Ing. (FH) Elektrotechnik
//DATUM: 10/2008
//INTERNET: www.maagic7.de
//
//AENDERUNGSVERMERKE:
//--------------------------------------------------------------------------------
//DATUM        NAME        AENDERUNG
//--------------------------------------------------------------------------------
//01.04.2020   S.Maag      Anzeige aktiver Kanal (DSP_CHANNEL).
//                         RETURN NullAny, wenn kein Kanal ausgewählt
//                         ENABLE wie bei WerteMultiplexern
//hinzugefügt---------------------------------------------------------------------
//-----------
//
//HINWEISE:
AUTHOR : 'S.Maag'
FAMILY : Maagic7
VERSION : 0.1


VAR_INPUT
  S1 : BOOL ;	//Select no. 1
  S2 : BOOL ;	//Select no. 2
  S3 : BOOL ;	//Select no. 3
  S4 : BOOL ;	//Select no. 4
  ENABLE : BOOL ;	//If not Enabled: RET_VAL:=NullAny
  ANY1 : ANY ;	//ANY Pointer 1
  ANY2 : ANY ;	//ANY Pointer 3
  ANY3 : ANY ;	//ANY Pointer 3
  ANY4 : ANY ;	//ANY Pointer 4
END_VAR
VAR_OUTPUT
  DSP_CHANNEL : INT ;	//Displays the activated channel
END_VAR
VAR_TEMP
  anyNull : ANY ;
END_VAR
BEGIN
NETWORK
TITLE =
//It isn't recomended to restore AR1 & AR2, it will be done automatically by the
//systems CALL operation, when leaving the Function
      UN    #ENABLE; // keine Freigabe, dann 0 ausgeben
      SPB   OFF;

